CASE units OF
    AxesMoveProcessWidgetUnits.ARCMINUTES:
        unitsText := '$'';
        aziDeg := field_azi_decimal / 60.0;
        eleDeg := field_ele_decimal / 60.0;
        rocDeg := field_roc_decimal / 60.0;
        ronDeg := field_ron_decimal / 60.0;
    AxesMoveProcessWidgetUnits.ARCSECCONDS:
        unitsText := '"';
        aziDeg := field_azi_decimal / 3600.0;
        eleDeg := field_ele_decimal / 3600.0;
        rocDeg := field_roc_decimal / 3600.0;
        ronDeg := field_ron_decimal / 3600.0;
    AxesMoveProcessWidgetUnits.DEGMINSEC:
        unitsText := '';
        aziDeg := DMS_TO_DEG(
            positive := field_azi_sign = AxesDialogSign.DIALOG_PLUS,
            degrees  := field_azi_d,
            minutes  := field_azi_m,
            seconds  := field_azi_s);
        eleDeg := DMS_TO_DEG(
            positive := field_ele_sign = AxesDialogSign.DIALOG_PLUS,
            degrees  := field_ele_d,
            minutes  := field_ele_m,
            seconds  := field_ele_s);
        rocDeg := DMS_TO_DEG(
            positive := field_roc_sign = AxesDialogSign.DIALOG_PLUS,
            degrees  := field_roc_d,
            minutes  := field_roc_m,
            seconds  := field_roc_s);
        ronDeg := DMS_TO_DEG(
            positive := field_ron_sign = AxesDialogSign.DIALOG_PLUS,
            degrees  := field_ron_d,
            minutes  := field_ron_m,
            seconds  := field_ron_s);
    AxesMoveProcessWidgetUnits.DEGREES:
        unitsText := '°';
        aziDeg := field_azi_decimal;
        eleDeg := field_ele_decimal;
        rocDeg := field_roc_decimal;
        ronDeg := field_ron_decimal;
    AxesMoveProcessWidgetUnits.RADIANS:
        unitsText := 'rad';
        aziDeg := RAD_TO_DEG(field_azi_decimal);
        eleDeg := RAD_TO_DEG(field_ele_decimal);
        rocDeg := RAD_TO_DEG(field_roc_decimal);
        ronDeg := RAD_TO_DEG(field_ron_decimal);
END_CASE

END_FUNCTION_BLOCK

// ---- MTCS/Axes/Widgets/AxesManualMoveVelocityWidget.TcPOU
FUNCTION_BLOCK AxesManualMoveVelocityWidget
VAR_INPUT
    field_alphaVelocity : LREAL;
    field_deltaVelocity : LREAL;
    field_units : AxesMoveVelocityUnits;
    label_units : STRING;
    do_start : BOOL;
    do_stop : BOOL;
    
    setAlphaDeltaVelocityStatus : StatusWidget;
END_VAR
VAR_OUTPUT
    alphaTravelledSoFar : AxesAlphaWidget;
    deltaTravelledSoFar : AxesDeltaWidget;
    alphaPerMinute : AxesAlphaWidget;
    deltaPerMinute : AxesDeltaWidget;
END_VAR
VAR_IN_OUT
    ref : Axes;
END_VAR
VAR
END_VAR


setAlphaDeltaVelocityStatus(
    text  := ref.processes.setAlphaDeltaVelocity.actualStatus,
    color := HealthBusyToColor(healthStatus := ref.processes.setAlphaDeltaVelocity.statuses.healthStatus, 
                               busyStatus   := ref.processes.setAlphaDeltaVelocity.statuses.busyStatus));

label_units := AxesMoveVelocityUnitsToString(field_units);
                      
alphaTravelledSoFar(radians := ref.target.alphaTravelled.radians.value);
deltaTravelledSoFar(radians := ref.target.deltaTravelled.radians.value);

alphaPerMinute(radians := ref.target.alphaVelocity.radiansPerSecond.value * 60.0);
deltaPerMinute(radians := ref.target.deltaVelocity.radiansPerSecond.value * 60.0);

IF do_start THEN
    ref.processes.setAlphaDeltaVelocity.request( units := field_units, alphaVelocity := field_alphaVelocity, deltaVelocity := field_deltaVelocity);
    do_start := FALSE;
END_IF

IF do_stop THEN
    ref.processes.setAlphaDeltaVelocity.request( units := AxesMoveVelocityUnits.ARCSECONDS_PER_SECOND, alphaVelocity := 0.0, deltaVelocity := 0.0);
    do_stop := FALSE;
END_IF

END_FUNCTION_BLOCK

// ---- MTCS/Axes/Widgets/AxesManualPositionsWidget.TcPOU
FUNCTION_BLOCK AxesManualPositionsWidget
VAR_INPUT
END_VAR
VAR_OUTPUT
    invisiblePosition0 : BOOL;
    invisiblePosition1 : BOOL;
    invisiblePosition2 : BOOL;
    invisiblePosition3 : BOOL;
    invisiblePosition4 : BOOL;
    invisiblePosition5 : BOOL;
    invisiblePosition6 : BOOL;
    invisiblePosition7 : BOOL;
    invisiblePosition8 : BOOL;
    invisiblePosition9 : BOOL;
    invisiblePosition10 : BOOL;
    invisiblePosition11 : BOOL;
    invisiblePosition12 : BOOL;
    invisiblePosition13 : BOOL;
    invisiblePosition14 : BOOL;
    invisiblePosition15 : BOOL;
    invisiblePosition16 : BOOL;
    invisiblePosition17 : BOOL;
    invisiblePosition18 : BOOL;
    invisiblePosition19 : BOOL;
END_VAR
VAR_IN_OUT
    ref : Axes;
    ref_operatorStatus : OperatorStatus;
END_VAR
VAR
END_VAR

invisiblePosition0 := NOT (ref.config.knownPositions.position0.allowObserver OR ref_operatorStatus.tech) OR ref.config.knownPositions.position0.name = '';
invisiblePosition1 := NOT (ref.config.knownPositions.position1.allowObserver OR ref_operatorStatus.tech) OR ref.config.knownPositions.position1.name = '';
invisiblePosition2 := NOT (ref.config.knownPositions.position2.allowObserver OR ref_operatorStatus.tech) OR ref.config.knownPositions.position2.name = '';
invisiblePosition3 := NOT (ref.config.knownPositions.position3.allowObserver OR ref_operatorStatus.tech) OR ref.config.knownPositions.position3.name = '';
invisiblePosition4 := NOT (ref.config.knownPositions.position4.allowObserver OR ref_operatorStatus.tech) OR ref.config.knownPositions.position4.name = '';
invisiblePosition5 := NOT (ref.config.knownPositions.position5.allowObserver OR ref_operatorStatus.tech) OR ref.config.knownPositions.position5.name = '';
invisiblePosition6 := NOT (ref.config.knownPositions.position6.allowObserver OR ref_operatorStatus.tech) OR ref.config.knownPositions.position6.name = '';
invisiblePosition7 := NOT (ref.config.knownPositions.position7.allowObserver OR ref_operatorStatus.tech) OR ref.config.knownPositions.position7.name = '';
invisiblePosition8 := NOT (ref.config.knownPositions.position8.allowObserver OR ref_operatorStatus.tech) OR ref.config.knownPositions.position8.name = '';
invisiblePosition9 := NOT (ref.config.knownPositions.position9.allowObserver OR ref_operatorStatus.tech) OR ref.config.knownPositions.position9.name = '';
invisiblePosition10 := NOT (ref.config.knownPositions.position10.allowObserver OR ref_operatorStatus.tech) OR ref.config.knownPositions.position10.name = '';
invisiblePosition11 := NOT (ref.config.knownPositions.position11.allowObserver OR ref_operatorStatus.tech) OR ref.config.knownPositions.position11.name = '';
invisiblePosition12 := NOT (ref.config.knownPositions.position12.allowObserver OR ref_operatorStatus.tech) OR ref.config.knownPositions.position12.name = '';
invisiblePosition13 := NOT (ref.config.knownPositions.position13.allowObserver OR ref_operatorStatus.tech) OR ref.config.knownPositions.position13.name = '';
invisiblePosition14 := NOT (ref.config.knownPositions.position14.allowObserver OR ref_operatorStatus.tech) OR ref.config.knownPositions.position14.name = '';
invisiblePosition15 := NOT (ref.config.knownPositions.position15.allowObserver OR ref_operatorStatus.tech) OR ref.config.knownPositions.position15.name = '';
invisiblePosition16 := NOT (ref.config.knownPositions.position16.allowObserver OR ref_operatorStatus.tech) OR ref.config.knownPositions.position16.name = '';
invisiblePosition17 := NOT (ref.config.knownPositions.position17.allowObserver OR ref_operatorStatus.tech) OR ref.config.knownPositions.position17.name = '';
invisiblePosition18 := NOT (ref.config.knownPositions.position18.allowObserver OR ref_operatorStatus.tech) OR ref.config.knownPositions.position18.name = '';
invisiblePosition19 := NOT (ref.config.knownPositions.position19.allowObserver OR ref_operatorStatus.tech) OR ref.config.knownPositions.position19.name = '';

END_FUNCTION_BLOCK

// ---- MTCS/Axes/Widgets/AxesManualMoveAbsoluteWidget.TcPOU
FUNCTION_BLOCK AxesManualMoveAbsoluteWidget
VAR_INPUT
    moveAbsolute : AxesMultiMoveProcessWIdget;
END_VAR
VAR_OUTPUT
END_VAR
VAR_IN_OUT
    ref : Axes;
END_VAR
VAR
END_VAR

moveAbsolute(
    aziDisabled := ref.processes.moveAbsolute.statuses.enabledStatus.disabled OR ref.parts.azi.statuses.poweredStatus.disabled,
    eleDisabled := ref.processes.moveAbsolute.statuses.enabledStatus.disabled OR ref.parts.ele.statuses.poweredStatus.disabled,
    rocDisabled := ref.processes.moveAbsolute.statuses.enabledStatus.disabled OR ref.parts.roc.statuses.poweredStatus.disabled,
    ronDisabled := ref.processes.moveAbsolute.statuses.enabledStatus.disabled OR ref.parts.ron.statuses.poweredStatus.disabled,
    process := ref.processes.moveAbsolute,  
    title := 'Move absolute');

END_FUNCTION_BLOCK

// ---- MTCS/Axes/Widgets/AxesElevationAxisWidget.TcPOU
FUNCTION_BLOCK AxesElevationAxisWidget
VAR_INPUT
    activeTab : AxesElevationAxisTabs;
END_VAR
VAR_OUTPUT
END_VAR
VAR_IN_OUT
    ref : AxesElevationAxis;
    ref_driveChannel : AX52XXDriveChannel;
END_VAR
VAR
	actualStatus : StatusWidget;
    
    processes_powerOnStatus : StatusWidget;
    processes_powerOffStatus : StatusWidget;
    processes_resetStatus : StatusWidget;
    processes_doHomingStatus : StatusWidget;
    processes_unlockBrakeStatus : StatusWidget;
    processes_stopStatus : StatusWidget;
    processes_moveAbsoluteStatus : StatusWidget;
    processes_moveRelativeStatus : StatusWidget;
    processes_moveVelocityStatus : StatusWidget;
    processes_moveOutOfLimitSwitchStatus : StatusWidget;
    
    lidaCommonHealthStatus : HealthStatus;
    lidaCommonBusyStatus   : BusyStatus;
    lidaCommonStatusColor  : StatusColor;
    
    processCommonHealthStatus : HealthStatus;
    processCommonBusyStatus   : BusyStatus;
    processCommonStatusColor  : StatusColor;
    
    
    button_overview         : SubSubSystemButtonWidget('Overview'           , AxesElevationAxisTabs.OVERVIEW);
    button_processes        : SubSubSystemButtonWidget('Processes'          , AxesElevationAxisTabs.PROCESSES);
    button_driveChannel     : SubSubSystemButtonWidget('Drive channel'      , AxesElevationAxisTabs.DRIVE_CHANNEL);   
    button_virtualAxis      : SubSubSystemButtonWidget('Virtual axis'       , AxesElevationAxisTabs.VIRTUAL_AXIS);  
    button_physicalAxis     : SubSubSystemButtonWidget('Physical axis'      , AxesElevationAxisTabs.PHYSICAL_AXIS);  
    button_lidas            : SubSubSystemButtonWidget('LIDAs'              , AxesElevationAxisTabs.LIDAS);
    button_absoluteEncoder  : SubSubSystemButtonWidget('Absolute encoder'   , AxesElevationAxisTabs.ABSOLUTE_ENCODER);
    
    driveChannel    : AX52XXDriveChannelWidget;
    virtualAxis     : AngularAxisWidget;
    physicalAxis    : AngularAxisWidget;
    
    lida1 : IncrementalEncoderWidget;
    lida2 : IncrementalEncoderWidget;
    
    actPos : AxesAngleWidget;
    setPos : AxesAngleWidget;
    targetPos : AxesAngleWidget;
END_VAR


actualStatus(text  := ref.actualStatus,
             color := HealthBusyToColor(healthStatus := ref.statuses.healthStatus, 
                                        busyStatus   := ref.statuses.busyStatus));

processes_powerOffStatus(
    text  := ref.processes.powerOff.actualStatus,
    color := HealthBusyToColor(healthStatus := ref.processes.powerOff.statuses.healthStatus, 
                               busyStatus   := ref.processes.powerOff.statuses.busyStatus));
processes_powerOnStatus(
    text  := ref.processes.powerOn.actualStatus,
    color := HealthBusyToColor(healthStatus := ref.processes.powerOn.statuses.healthStatus, 
                               busyStatus   := ref.processes.powerOn.statuses.busyStatus));
processes_resetStatus(
    text  := ref.processes.reset.actualStatus,
    color := HealthBusyToColor(healthStatus := ref.processes.reset.statuses.healthStatus, 
                               busyStatus   := ref.processes.reset.statuses.busyStatus));
processes_doHomingStatus(
    text  := ref.processes.doHoming.actualStatus,
    color := HealthBusyToColor(healthStatus := ref.processes.doHoming.statuses.healthStatus, 
                               busyStatus   := ref.processes.doHoming.statuses.busyStatus));
processes_unlockBrakeStatus(
    text  := ref.processes.unlockBrake.actualStatus,
    color := HealthBusyToColor(healthStatus := ref.processes.unlockBrake.statuses.healthStatus, 
                               busyStatus   := ref.processes.unlockBrake.statuses.busyStatus));
processes_stopStatus(
    text  := ref.processes.stop.actualStatus,
    color := HealthBusyToColor(healthStatus := ref.processes.stop.statuses.healthStatus, 
                               busyStatus   := ref.processes.stop.statuses.busyStatus));
processes_moveAbsoluteStatus(
    text  := ref.processes.moveAbsolute.actualStatus,
    color := HealthBusyToColor(healthStatus := ref.processes.moveAbsolute.statuses.healthStatus, 
                               busyStatus   := ref.processes.moveAbsolute.statuses.busyStatus));
processes_moveRelativeStatus(
    text  := ref.processes.moveRelative.actualStatus,
    color := HealthBusyToColor(healthStatus := ref.processes.moveRelative.statuses.healthStatus, 
                               busyStatus   := ref.processes.moveRelative.statuses.busyStatus));
processes_moveVelocityStatus(
    text  := ref.processes.moveVelocity.actualStatus,
    color := HealthBusyToColor(healthStatus := ref.processes.moveVelocity.statuses.healthStatus, 
                               busyStatus   := ref.processes.moveVelocity.statuses.busyStatus));
processes_moveOutOfLimitSwitchStatus(
    text  := ref.processes.moveOutOfLimitSwitch.actualStatus,
    color := HealthBusyToColor(healthStatus := ref.processes.moveOutOfLimitSwitch.statuses.healthStatus, 
                               busyStatus   := ref.processes.moveOutOfLimitSwitch.statuses.busyStatus));


driveChannel(ref := ref_driveChannel, name := 'ELE (Drive ELED channel A)');
virtualAxis(baseRef := ref.parts.virtualAxis, ref := ref.parts.virtualAxis);
physicalAxis(baseRef := ref.parts.physicalAxis, ref := ref.parts.physicalAxis);                


lidaCommonHealthStatus(
     isGood :=      ref.parts.lida1.statuses.healthStatus.isGood 
                AND ref.parts.lida2.statuses.healthStatus.isGood,
     hasWarning :=  ref.parts.lida1.statuses.healthStatus.hasWarning 
                 OR ref.parts.lida2.statuses.healthStatus.hasWarning);

lidaCommonBusyStatus(
    isBusy :=      ref.parts.lida1.statuses.busyStatus.isBusy 
                OR ref.parts.lida2.statuses.busyStatus.isBusy);

lidaCommonStatusColor := HealthBusyToColor(healthStatus := lidaCommonHealthStatus, busyStatus := lidaCommonBusyStatus);


processCommonHealthStatus(
     isGood :=      ref.processes.powerOn.statuses.healthStatus.isGood 
                AND ref.processes.powerOff.statuses.healthStatus.isGood
                AND ref.processes.reset.statuses.healthStatus.isGood
                AND ref.processes.doHoming.statuses.healthStatus.isGood
                AND ref.processes.unlockBrake.statuses.healthStatus.isGood
                AND ref.processes.stop.statuses.healthStatus.isGood
                AND ref.processes.moveAbsolute.statuses.healthStatus.isGood
                AND ref.processes.moveRelative.statuses.healthStatus.isGood
                AND ref.processes.moveVelocity.statuses.healthStatus.isGood
                AND ref.processes.moveOutOfLimitSwitch.statuses.healthStatus.isGood,
     hasWarning :=  ref.processes.powerOn.statuses.healthStatus.hasWarning 
                 OR ref.processes.powerOff.statuses.healthStatus.hasWarning
                 OR ref.processes.reset.statuses.healthStatus.hasWarning
                 OR ref.processes.doHoming.statuses.healthStatus.hasWarning
                 OR ref.processes.unlockBrake.statuses.healthStatus.hasWarning
                 OR ref.processes.stop.statuses.healthStatus.hasWarning
                 OR ref.processes.moveAbsolute.statuses.healthStatus.hasWarning
                 OR ref.processes.moveRelative.statuses.healthStatus.hasWarning
                 OR ref.processes.moveVelocity.statuses.healthStatus.hasWarning
                 OR ref.processes.moveOutOfLimitSwitch.statuses.healthStatus.hasWarning);

processCommonBusyStatus(
    isBusy :=      ref.processes.powerOn.statuses.busyStatus.busy 
                 OR ref.processes.powerOff.statuses.busyStatus.busy
                 OR ref.processes.reset.statuses.busyStatus.busy
                 OR ref.processes.doHoming.statuses.busyStatus.busy
                 OR ref.processes.unlockBrake.statuses.busyStatus.busy
                 OR ref.processes.stop.statuses.busyStatus.busy
                 OR ref.processes.moveAbsolute.statuses.busyStatus.busy
                 OR ref.processes.moveRelative.statuses.busyStatus.busy
                 OR ref.processes.moveVelocity.statuses.busyStatus.busy
                 OR ref.processes.moveOutOfLimitSwitch.statuses.busyStatus.busy);

processCommonStatusColor := HealthBusyToColor(healthStatus := processCommonHealthStatus, busyStatus := processCommonBusyStatus);
     

lida1(ref := ref.parts.lida1);
lida2(ref := ref.parts.lida2);

button_overview(        color := actualStatus.color                     , activeTab := activeTab);
button_processes(       color := processCommonStatusColor               , activeTab := activeTab);
button_driveChannel(    color := driveChannel.actualStatus.color        , activeTab := activeTab);
button_virtualAxis(     color := virtualAxis.base.actualStatus.color    , activeTab := activeTab);
button_physicalAxis(    color := physicalAxis.base.actualStatus.color   , activeTab := activeTab);
button_lidas(           color := lidaCommonStatusColor                  , activeTab := activeTab);
button_absoluteEncoder( color := HealthToColor(ref.parts.absoluteEncoder.statuses.healthStatus), activeTab := activeTab);

actPos(degrees := ref.actPos.degrees.value, format := '%d° %.2d$' %04.1f"', showPlus := FALSE, showMinus := TRUE);
setPos(degrees := ref.setPos.degrees.value, format := '%d° %.2d$' %04.1f"', showPlus := FALSE, showMinus := TRUE);
targetPos(degrees := ref.targetPos.degrees.value, format := '%d° %.2d$' %04.1f"', showPlus := FALSE, showMinus := TRUE);

END_FUNCTION_BLOCK

// ---- MTCS/Common/Widgets/SubSubSystemButtonWidget.TcPOU
FUNCTION_BLOCK SubSubSystemButtonWidget EXTENDS SubSystemButtonWidget
VAR_INPUT
END_VAR
VAR_IN_OUT
END_VAR
VAR_OUTPUT
END_VAR
VAR
END_VAR

SUPER^(activeTab := activeTab);

END_FUNCTION_BLOCK

// ---- MTCS/Common/Widgets/SubSystemButtonWidget.TcPOU
FUNCTION_BLOCK SubSystemButtonWidget
VAR_INPUT
    color : StatusColor;
    hideColor : BOOL := FALSE;
END_VAR
VAR_IN_OUT
    activeTab : INT;
END_VAR
VAR_OUTPUT
    name : STRING;
    thisTab : INT;
    colorVisible : BOOL;
    
    activated : BOOL;
    notActivated : BOOL;
    
    isNotGreen : BOOL;
    isNotRed : BOOL;
    isNotBlue : BOOL;
    isNotOrange : BOOL;
    isNotGray : BOOL;
END_VAR
VAR
    do_activate : BOOL;
END_VAR


IF do_activate THEN
    activeTab := thisTab;
    do_activate := FALSE;
END_IF

activated := activeTab = thisTab;
notActivated := NOT activated;

isNotRed    := color.bg <> Colors.RED;
isNotBlue   := color.bg <> Colors.BLUE;
isNotOrange := color.bg <> Colors.ORANGE;
isNotGray   := color.bg <> Colors.GRAY;
isNotGreen  := color.bg <> Colors.GREEN;

METHOD FB_init : BOOL
VAR_INPUT
	bInitRetains : BOOL; // if TRUE, the retain variables are initialized (warm start / cold start)
	bInCopyCode : BOOL;  // if TRUE, the instance afterwards gets moved into the copy code (online change)
    n : STRING;
    tab : INT;
END_VAR
name := n;
thisTab := tab;
END_METHOD

END_FUNCTION_BLOCK

// ---- MTCS/Common/Widgets/AX52XXDriveChannelWidget.TcPOU
FUNCTION_BLOCK AX52XXDriveChannelWidget
VAR_INPUT
    name : STRING;
END_VAR
VAR_OUTPUT
	actualStatus : StatusWidget;
    
    input0 : BOOL;
    input1 : BOOL;
    input2 : BOOL;
    input3 : BOOL;
    input4 : BOOL;
    input5 : BOOL;
    input6 : BOOL;
    input7 : BOOL;
    
    output0 : BOOL;
    output1 : BOOL;
    output2 : BOOL;
    output3 : BOOL;
    output4 : BOOL;
    output5 : BOOL;
    output6 : BOOL;
    output7 : BOOL;
    
	processes_setBrakeStatus : StatusWidget;
	processes_acknowledgeSafetyError : StatusWidget;
END_VAR
VAR
END_VAR
VAR_IN_OUT
	ref : AX52XXDriveChannel;
END_VAR


actualStatus(text  := ref.actualStatus,
             color := HealthBusyToColor(healthStatus := ref.statuses.healthStatus, 
                                        busyStatus   := ref.statuses.busyStatus));
                                        
input0 := ref.digitalInputs.0;          
input1 := ref.digitalInputs.1;          
input2 := ref.digitalInputs.2;          
input3 := ref.digitalInputs.3;          
input4 := ref.digitalInputs.4;          
input5 := ref.digitalInputs.5;          
input6 := ref.digitalInputs.6;          
input7 := ref.digitalInputs.7;
      
output0 := ref.digitalOutputs.0;
output1 := ref.digitalOutputs.1;
output2 := ref.digitalOutputs.2;
output3 := ref.digitalOutputs.3;
output4 := ref.digitalOutputs.4;
output5 := ref.digitalOutputs.5;
output6 := ref.digitalOutputs.6;
output7 := ref.digitalOutputs.7;

processes_setBrakeStatus(text  := ref.processes.setBrake.actualStatus,
                         color := HealthBusyToColor(healthStatus := ref.processes.setBrake.statuses.healthStatus, 
                                                    busyStatus   := ref.processes.setBrake.statuses.busyStatus));
processes_acknowledgeSafetyError(text  := ref.processes.acknowledgeSafetyError.actualStatus,
                         color := HealthBusyToColor(healthStatus := ref.processes.acknowledgeSafetyError.statuses.healthStatus, 
                                                    busyStatus   := ref.processes.acknowledgeSafetyError.statuses.busyStatus));

END_FUNCTION_BLOCK

// ---- MTCS/Common/Widgets/AngularAxisWidget.TcPOU
FUNCTION_BLOCK AngularAxisWidget
VAR_INPUT
END_VAR
VAR_OUTPUT
    positionSymbol : STRING := '°';
    velocitySymbol : STRING := '°/s';
    base : BaseAxisWidget;
END_VAR
VAR_IN_OUT
    baseRef : AngularAxis;
    ref : AngularAxis;
END_VAR
VAR
END_VAR

base(ref := baseRef);

END_FUNCTION_BLOCK

// ---- MTCS/Common/Widgets/BaseAxisWidget.TcPOU
FUNCTION_BLOCK BaseAxisWidget
VAR_INPUT
END_VAR
VAR_OUTPUT
    coupled : BOOL;
    decoupled : BOOL;
	(* widgets *)
	moveAbsoluteProcess : McProcessWidget;
	moveVelocityProcess : McProcessWidget;
	actualStatus : StatusWidget;
END_VAR
VAR_IN_OUT
    ref : BaseAxis;
END_VAR
VAR
END_VAR


coupled := ref.axis_ref.Status.Coupled;
decoupled := NOT coupled;

// update the widgets
moveAbsoluteProcess(process := ref.processes.moveAbsolute);
moveVelocityProcess(process := ref.processes.moveVelocity);
actualStatus(text  := ref.actualStatus,
             color := HealthBusyToColor(healthStatus := ref.statuses.healthStatus, 
                                        busyStatus   := ref.statuses.busyStatus));

END_FUNCTION_BLOCK

// ---- MTCS/Common/Widgets/McProcessWidget.TcPOU
FUNCTION_BLOCK McProcessWidget
VAR_INPUT
END_VAR
VAR_OUTPUT
    actualStatus : StatusWidget;
END_VAR
VAR_IN_OUT
	process : BaseMcProcess;
END_VAR
VAR
END_VAR

actualStatus(text  := process.actualStatus,
             color := HealthBusyToColor(healthStatus := process.statuses.healthStatus,
                                        busyStatus   := process.statuses.busyStatus));

END_FUNCTION_BLOCK

// ---- MTCS/Common/StateMachines/BaseMcProcess.TcPOU
FUNCTION_BLOCK BaseMcProcess EXTENDS SM_BaseMcProcess
VAR_INPUT
END_VAR
VAR_OUTPUT
END_VAR
VAR
	testVar3 : BOOL;
END_VAR

SUPER^();
                                  
IF statuses.healthStatus.good THEN

	IF statuses.busyStatus.idle THEN
		actualStatus := 'Idle';
	ELSIF statuses.busyStatus.busy THEN
		actualStatus := 'Busy';
	ELSE
		actualStatus := '';
	END_IF;

ELSIF statuses.healthStatus.bad THEN
	
	IF statuses.busyStatus.idle THEN
		IF errorId = 0 THEN
			actualStatus := 'Error';
		ELSE
			actualStatus := CONCAT(CONCAT('Error (', UDINT_TO_STRING(errorId)), ')');
		END_IF
	ELSIF statuses.busyStatus.busy THEN
		IF errorId = 0 THEN
			actualStatus := 'Busy and error';
		ELSE
			actualStatus := CONCAT(CONCAT('Busy and error (', UDINT_TO_STRING(errorId)), ')');
		END_IF
	ELSE
		IF errorId = 0 THEN
			actualStatus := 'Error';
		ELSE
			actualStatus := CONCAT(CONCAT('Error (', UDINT_TO_STRING(errorId)), ')');
		END_IF
	END_IF;

ELSE
	actualStatus := '';
END_IF;

END_FUNCTION_BLOCK

// ---- MTCS/Common/StateMachines/BaseAxis.TcPOU
FUNCTION_BLOCK BaseAxis EXTENDS SM_BaseAxis
VAR_INPUT
END_VAR
VAR_OUTPUT
END_VAR
VAR
	_mc_moveAbsolute1         : MC_MoveAbsolute;
	_mc_moveAbsolute2         : MC_MoveAbsolute;
    _moveAbsoluteAlternator   : BOOL;
    _previousMoveAbsolutePosition : LREAL;
    _previousMoveAbsoluteMaxVelocity : LREAL;
    _moveAbsoluteStopping   : BOOL;
    _mc_moveVelocity : MC_MoveVelocity;
    _mc_moveRelative : MC_MoveRelative;
    
	_mc_power : MC_Power;
	_mc_reset : MC_Reset;
	_mc_halt : MC_Halt;
	_mc_halt2 : MC_Halt;
	_mc_gearIn : MC_GearIn;
	_mc_gearOut : MC_GearOut;
    _mc_setPosition : MC_SetPosition;
    _mc_extSetPointGenEnable : MC_ExtSetPointGenEnable;
    _mc_extSetPointGenDisable : MC_ExtSetPointGenDisable;
    _mc_home : MC_Home;
    _mc_jog : MC_Jog;
    
	_powered : BOOL;
    
    _masterAddr : POINTER TO AXIS_REF := 0;
    
    _ctrl_pi_params : ST_CTRL_PI_PARAMS;
    _ctrl_pi : FB_CTRL_PI;
    _mc_moveVelocity1 : MC_MoveVelocity;
    _mc_moveVelocity2 : MC_MoveVelocity;
    
    _mc_writeParameter : MC_WriteParameter;
    _mc_writeBoolParameter : MC_WriteBoolParameter;
    _mc_readParameter : MC_ReadParameter;
    _mc_readBoolParameter : MC_ReadBoolParameter;
    
    
    Kp : LREAL := 1.0;
    Td : LREAL := 0.0;
END_VAR

SUPER^.axis_ref.ReadStatus();

_update();

// command the axis
_powering();
_movingAbsolute();
_movingRelative();
_resetting();
_initializing();
_stopping();
_stoppingParametrized();
_gearIn();
_gearOut();
_setPosition();
_moveVelocity();
_enableExtSetGen();
_disableExtSetGen();
_forceCalibration();
_resetCalibration();

_readParameter();
_readBoolParameter();
_writeParameter();
_writeBoolParameter();

_update();

METHOD _forceCalibration
VAR_INPUT
END_VAR

_mc_home(
    Execute     := processes.forceCalibration.statuses.busyStatus.busy,
    Position    := 0.0,
    HomingMode  := MC_HomingMode.MC_ForceCalibration,
    Axis        := axis_ref);

(* update the health status *)
SUPER^.processes.forceCalibration.statuses.healthStatus(isGood := NOT _mc_home.Error);

(* update the busy status *)
SUPER^.processes.forceCalibration.statuses.busyStatus(isBusy := _mc_home.Busy);

(* update the error ID *)
SUPER^.processes.forceCalibration.errorId := _mc_home.ErrorId;
END_METHOD

METHOD _movingAbsolute
VAR_INPUT
END_VAR
IF processes.moveAbsolute.statuses.busyStatus.busy THEN
	
    // MC_MoveAbsolute is a single command to instruct the axis to go to some position.
    // This position cannot be changed later: the command only does what you initially requested
    // (in other words: it only uses the position at the time of the Execute trigger).
    
    // We don' t want this behaviour, as we would like to be able to change the setpoint
    // position also during positioning. There are many use cases for this behaviour, e.g.:
    //  - you can send corrections to the axis while the position loop is running
    //  - you can change your mind while the positioning is running.
    
    // Therefore, we need 2 MC_MoveAbsolute commands, that abort each other alternatingly.
    // At each PLC cycle, one MC_MoveAbsolute command will be Busy and the other will be
    // CommandAborted. Only when one of them is Done (or Error), the motion has ended.
    
    IF    _previousMoveAbsolutePosition <> processes.moveAbsolute.get.position 
       OR _previousMoveAbsoluteMaxVelocity <> processes.moveAbsolute.get.maxVelocity
    THEN
        _moveAbsoluteAlternator := NOT _moveAbsoluteAlternator;
        _previousMoveAbsolutePosition := processes.moveAbsolute.get.position;
        _previousMoveAbsoluteMaxVelocity := processes.moveAbsolute.get.maxVelocity;
	END_IF
    
    IF _moveAbsoluteAlternator THEN
    
        _mc_moveAbsolute2(Axis := axis_ref, Execute := FALSE);
        
        _mc_moveAbsolute1(
            Axis       := axis_ref,
            Execute    := TRUE,
            Position   := processes.moveAbsolute.get.position,
            Velocity   := processes.moveAbsolute.get.maxVelocity,
            BufferMode := MC_BufferMode.MC_Aborting);
        
        (* update the statuses *)
        processes.moveAbsolute.statuses.healthStatus(isGood := NOT _mc_moveAbsolute1.Error);
        processes.moveAbsolute.errorId := _mc_moveAbsolute1.ErrorId;
        processes.moveAbsolute.statuses.busyStatus(isBusy := _mc_moveAbsolute1.Busy);
    ELSE
        
        _mc_moveAbsolute1(Axis := axis_ref, Execute := FALSE);
        
        _mc_moveAbsolute2(
            Axis       := axis_ref,
            Execute    := TRUE,
            Position   := processes.moveAbsolute.get.position,
            Velocity   := processes.moveAbsolute.get.maxVelocity,
            BufferMode := MC_BufferMode.MC_Aborting);
        
        (* update the statuses *)
        processes.moveAbsolute.statuses.healthStatus(isGood := NOT _mc_moveAbsolute2.Error);
        processes.moveAbsolute.errorId := _mc_moveAbsolute2.ErrorId;
        processes.moveAbsolute.statuses.busyStatus(isBusy := _mc_moveAbsolute2.Busy);
        
	END_IF
	
    (* reset the function blocks if needed *)
    IF processes.moveAbsolute.statuses.busyStatus.idle THEN
        _mc_moveAbsolute1(Axis := axis_ref, Execute := FALSE);
        _mc_moveAbsolute2(Axis := axis_ref, Execute := FALSE);
	END_IF
    
END_IF
END_METHOD

METHOD _writeBoolParameter
VAR_INPUT
END_VAR

_mc_writeBoolParameter(
    Execute         := processes.writeBoolParameter.statuses.busyStatus.busy,
    ParameterNumber := processes.writeBoolParameter.get.parameterNumber,
    Value           := processes.writeBoolParameter.get.value,
    Axis            := axis_ref);

(* update the health status *)
SUPER^.processes.writeBoolParameter.statuses.healthStatus(isGood := NOT _mc_writeBoolParameter.Error);

(* update the busy status *)
SUPER^.processes.writeBoolParameter.statuses.busyStatus(isBusy := _mc_writeBoolParameter.Busy);

(* update the error ID *)
SUPER^.processes.writeBoolParameter.errorId := _mc_writeBoolParameter.ErrorId;
END_METHOD

METHOD _gearIn
VAR_INPUT
END_VAR

IF _masterAddr = 0 THEN
    processes.gearIn.setBad();
    processes.gearIn.setFinished();
ELSE
    _mc_gearIn(
        Execute := processes.gearIn.statuses.busyStatus.busy,
        Master  := _masterAddr^,
        Slave   := axis_ref);
    
    (* update the health status *)
    SUPER^.processes.gearIn.statuses.healthStatus(isGood := NOT _mc_gearIn.Error);
    
    (* update the busy status *)
    SUPER^.processes.gearIn.statuses.busyStatus(isBusy := _mc_gearIn.Busy);
    
    (* update the error ID *)
    SUPER^.processes.gearIn.errorId := _mc_gearIn.ErrorId;
END_IF
END_METHOD

METHOD _moveVelocity
VAR_INPUT
END_VAR

IF processes.moveVelocity.isBusy() THEN
    
    IF NOT processes.moveVelocity.isStarted() THEN
        IF processes.moveVelocity.get.value >= 0 THEN
            _mc_moveVelocity(Execute := FALSE, Axis := axis_ref);
            _mc_moveVelocity(
                Execute      := TRUE,
                Velocity     := ABS(processes.moveVelocity.get.value),
                Acceleration := 0,
                Deceleration := 0,
                Jerk         := 0,
                Direction    := MC_Positive_Direction,
                Axis         := axis_ref);
        ELSE
            _mc_moveVelocity(Execute := FALSE, Axis := axis_ref);
            _mc_moveVelocity(
                Execute      := TRUE,
                Velocity     := ABS(processes.moveVelocity.get.value),
                Acceleration := 0,
                Deceleration := 0,
                Jerk         := 0,
                Direction    := MC_Negative_Direction,
                Axis         := axis_ref);
        END_IF
        processes.moveVelocity.setStarted();
    ELSE
        _mc_moveVelocity(Execute := FALSE, Axis := axis_ref);
	END_IF
    
    (* update the health status *)
    processes.moveVelocity.statuses.healthStatus(isGood := NOT _mc_moveVelocity.Error);
    
    (* update the busy status *)
    processes.moveVelocity.statuses.busyStatus(isBusy := _mc_moveVelocity.Busy AND NOT _mc_moveVelocity.InVelocity);
    
    (* update the error ID *)
    processes.moveVelocity.errorId := _mc_moveVelocity.ErrorId;
    
    
END_IF
END_METHOD

METHOD _readParameter
VAR_INPUT
END_VAR

_mc_readParameter(
    Enable          := processes.readParameter.statuses.busyStatus.busy,
    ParameterNumber := processes.readParameter.get.parameterNumber,
    Axis            := axis_ref,
    Value           => processes.readParameter.value);

(* update the health status *)
SUPER^.processes.readParameter.statuses.healthStatus(isGood := NOT _mc_readParameter.Error);

(* update the busy status *)
SUPER^.processes.readParameter.statuses.busyStatus(isBusy := _mc_readParameter.Busy);

(* update the error ID *)
SUPER^.processes.readParameter.errorId := _mc_readParameter.ErrorId;
END_METHOD

METHOD _stopping
VAR_INPUT
END_VAR

IF processes.stop.statuses.busyStatus.busy THEN
    
    _mc_halt(Execute := TRUE, Axis := axis_ref);
    
    IF _mc_halt.Error OR _mc_halt.Done OR _mc_halt.CommandAborted THEN
        _mc_halt(Execute := FALSE, Axis := axis_ref);
	END_IF
    
    (* update the health status *)
    SUPER^.processes.stop.statuses.healthStatus(isGood := NOT _mc_halt.Error);
    
    (* update the busy status *)
    SUPER^.processes.stop.statuses.busyStatus(isBusy := _mc_halt.Busy);
    
    (* update the error ID *)
    SUPER^.processes.stop.errorId := _mc_halt.ErrorId;
END_IF
END_METHOD

METHOD _resetCalibration
VAR_INPUT
END_VAR

_mc_home(
    Execute     := processes.resetCalibration.statuses.busyStatus.busy,
    Position    := 0.0,
    HomingMode  := MC_HomingMode.MC_ResetCalibration,
    Axis        := axis_ref);

(* update the health status *)
SUPER^.processes.resetCalibration.statuses.healthStatus(isGood := NOT _mc_home.Error);

(* update the busy status *)
SUPER^.processes.resetCalibration.statuses.busyStatus(isBusy := _mc_home.Busy);

(* update the error ID *)
SUPER^.processes.resetCalibration.errorId := _mc_home.ErrorId;
END_METHOD

METHOD _tracking_notworking
VAR_INPUT
END_VAR

VAR
    direction : MC_Direction;
END_VAR
IF processes.moveAbsolute.statuses.busyStatus.busy THEN
	
    IF NOT processes.moveAbsolute.isStarted() THEN
        _mc_moveVelocity1(Axis := axis_ref, Execute := FALSE);
        _mc_moveVelocity2(Axis := axis_ref, Execute := FALSE);
        _ctrl_pi_params.tCtrlCycleTime := GLOBAL.config.PLC_CTRL_TIME;
        _ctrl_pi_params.tTaskCycleTime := GLOBAL.config.PLC_TASK_TIME;
        processes.moveAbsolute.setStarted();
    END_IF

    _ctrl_pi_params.fKp := Kp;
    _ctrl_pi_params.tTn := LREAL_TO_TIME(Td); //ms
    _ctrl_pi_params.fOutMaxLimit :=  processes.moveAbsolute.get.maxVelocity;
    _ctrl_pi_params.fOutMinLimit := -processes.moveAbsolute.get.maxVelocity;
    
    _ctrl_pi(
        fSetpointValue := processes.moveAbsolute.get.position,
        fActualValue   := axis_ref.NcToPlc.ActPos,
        fManSyncValue  := 0.0,
        bSync          := FALSE,
        eMode          := eCTRL_MODE_ACTIVE,
        bHold          := FALSE,
        stParams       := _ctrl_pi_params);
    
    IF _ctrl_pi.fOut > 0 THEN
        direction := MC_Positive_Direction;
    ELSE
        direction := MC_Negative_Direction;
	END_IF
    
    _moveAbsoluteAlternator := NOT _moveAbsoluteAlternator;
    
    _moveAbsoluteStopping := ABS(processes.moveAbsolute.get.position - axis_ref.NcToPlc.ActPos) < 0.001
                             OR _mc_moveVelocity1.Error 
                             OR _mc_moveVelocity2.Error
                             OR (_mc_moveVelocity1.CommandAborted AND _mc_moveVelocity2.CommandAborted);
    
    IF _moveAbsoluteStopping THEN
        _mc_halt(Execute := TRUE, Axis := axis_ref);
        IF _mc_halt.Done THEN
            _mc_halt(Execute := FALSE, Axis := axis_ref);
            processes.moveAbsolute.setGood();
            processes.moveAbsolute.setFinished();
        ELSIF _mc_halt.Error OR _mc_halt.CommandAborted THEN
            _mc_halt(Execute := FALSE, Axis := axis_ref);
            processes.moveAbsolute.setBad();
            processes.moveAbsolute.setFinished();
		END_IF
    ELSIF _moveAbsoluteAlternator THEN
        _mc_moveVelocity2(Axis := axis_ref, Execute := FALSE);
        _mc_moveVelocity1(
            Execute      := TRUE,
            Velocity     := ABS(_ctrl_pi.fOut),
            Acceleration := 0,
            Deceleration := 0,
            Jerk         := 0,
            Direction    := direction,
            BufferMode := MC_BufferMode.MC_Aborting,
            Axis         := axis_ref);
            
            (* update the statuses *)
            //processes.moveAbsolute.statuses.busyStatus(isBusy := _mc_moveVelocity1.Busy);
            processes.moveAbsolute.statuses.healthStatus(isGood := NOT _mc_moveVelocity1.Error);
            processes.moveAbsolute.errorId := _mc_moveVelocity1.ErrorId;
    ELSE
        _mc_moveVelocity1(Axis := axis_ref, Execute := FALSE);
        _mc_moveVelocity2(
            Execute      := TRUE,
            Velocity     := ABS(_ctrl_pi.fOut),
            Acceleration := 0,
            Deceleration := 0,
            Jerk         := 0,
            Direction    := direction,
            BufferMode := MC_BufferMode.MC_Aborting,
            Axis         := axis_ref);
            
            (* update the statuses *)
            //processes.moveAbsolute.statuses.busyStatus(isBusy := _mc_moveVelocity2.Busy);
            processes.moveAbsolute.statuses.healthStatus(isGood := NOT _mc_moveVelocity2.Error);
            processes.moveAbsolute.errorId := _mc_moveVelocity2.ErrorId;
	END_IF
    
ELSE
    
    _ctrl_pi(eMode := eCTRL_MODE_RESET, stParams := _ctrl_pi_params);
    
END_IF
END_METHOD

METHOD _setPosition
VAR_INPUT
END_VAR

_mc_setPosition(
    Execute  := processes.setPosition.statuses.busyStatus.busy,
    Position := processes.setPosition.get.value,
    Mode     := FALSE,
    Axis     := axis_ref);

(* update the health status *)
SUPER^.processes.setPosition.statuses.healthStatus(isGood := NOT _mc_setPosition.Error);

(* update the busy status *)
SUPER^.processes.setPosition.statuses.busyStatus(isBusy := _mc_setPosition.Busy);

(* update the error ID *)
SUPER^.processes.setPosition.errorId := _mc_setPosition.ErrorId;
END_METHOD

METHOD _readBoolParameter
VAR_INPUT
END_VAR

_mc_readBoolParameter(
    Enable          := processes.readBoolParameter.statuses.busyStatus.busy,
    ParameterNumber := processes.readBoolParameter.get.parameterNumber,
    Axis            := axis_ref,
    Value           => processes.readBoolParameter.value);

(* update the health status *)
SUPER^.processes.readBoolParameter.statuses.healthStatus(isGood := NOT _mc_readBoolParameter.Error);

(* update the busy status *)
SUPER^.processes.readBoolParameter.statuses.busyStatus(isBusy := _mc_readBoolParameter.Busy);

(* update the error ID *)
SUPER^.processes.readBoolParameter.errorId := _mc_readBoolParameter.ErrorId;
END_METHOD

METHOD _update
VAR_INPUT
END_VAR
SUPER^();

IF statuses.healthStatus.good THEN
    IF statuses.busyStatus.idle THEN
        IF statuses.poweredStatus.enabled THEN
            actualStatus := 'Enabled';
        ELSIF statuses.poweredStatus.disabled THEN
            actualStatus := 'Disabled';
        ELSE
            actualStatus := 'Idle';
		END_IF
    ELSIF statuses.busyStatus.busy THEN
        IF statuses.motionStatus.forward THEN
            actualStatus := 'Moving forward';
        ELSIF statuses.motionStatus.backward THEN
            actualStatus := 'Moving backward';
        ELSIF statuses.motionStatus.standstill THEN
            actualStatus := 'Standing still';
        ELSE
            actualStatus := 'Busy';
		END_IF
    ELSE
        actualStatus := 'Good';
    END_IF
ELSIF statuses.healthStatus.bad THEN
    IF axis_ref.Status.ErrorId = 16992 THEN
        actualStatus := 'Controller not enabled!';
    ELSIF axis_ref.Status.ErrorId = 18000 THEN
        actualStatus := 'Drive not ready!';
    ELSE
        actualStatus := CONCAT(CONCAT('Error (id: ', UDINT_TO_STRING(axis_ref.Status.ErrorId)), ')');
	END_IF
ELSE
    actualStatus := '';
END_IF
END_METHOD

METHOD _enableExtSetGen
VAR_INPUT
END_VAR
_mc_extSetPointGenEnable(
	Axis    := axis_ref,
	Execute := processes.enableExtSetGen.statuses.busyStatus.busy);

(* update the health status *)
SUPER^.processes.enableExtSetGen.statuses.healthStatus(isGood := NOT _mc_extSetPointGenEnable.Error);

(* update the busy status *)
SUPER^.processes.enableExtSetGen.statuses.busyStatus(isBusy := _mc_extSetPointGenEnable.Busy);

(* update the error ID *)
SUPER^.processes.enableExtSetGen.errorId := _mc_extSetPointGenEnable.ErrorId;
END_METHOD

METHOD _initializing
VAR_INPUT
END_VAR
IF processes.initialize.statuses.busyStatus.busy THEN
    
	IF processes.initialize.statuses.startedStatus.notStarted THEN
		processes.reset.start();
		processes.initialize.setStarted();
	END_IF
    
    processes.initialize.statuses.busyStatus(isBusy := processes.reset.statuses.busyStatus.busy);
    processes.initialize.statuses.healthStatus(isGood := processes.reset.statuses.healthStatus.good);
    
    
ELSE
    // done
	processes.initialize.setFinished();
END_IF
END_METHOD

METHOD _disableExtSetGen
VAR_INPUT
END_VAR
_mc_extSetPointGenDisable(
	Axis    := axis_ref,
	Execute := processes.disableExtSetGen.statuses.busyStatus.busy);

(* update the health status *)
SUPER^.processes.disableExtSetGen.statuses.healthStatus(isGood := NOT _mc_extSetPointGenDisable.Error);

(* update the busy status *)
SUPER^.processes.disableExtSetGen.statuses.busyStatus(isBusy := _mc_extSetPointGenDisable.Busy);

(* update the error ID *)
SUPER^.processes.disableExtSetGen.errorId := _mc_extSetPointGenDisable.ErrorId;
END_METHOD

METHOD _writeParameter
VAR_INPUT
END_VAR

_mc_writeParameter(
    Execute         := processes.writeParameter.statuses.busyStatus.busy,
    ParameterNumber := processes.writeParameter.get.parameterNumber,
    Value           := processes.writeParameter.get.value,
    Axis            := axis_ref);

(* update the health status *)
SUPER^.processes.writeParameter.statuses.healthStatus(isGood := NOT _mc_writeParameter.Error);

(* update the busy status *)
SUPER^.processes.writeParameter.statuses.busyStatus(isBusy := _mc_writeParameter.Busy);

(* update the error ID *)
SUPER^.processes.writeParameter.errorId := _mc_writeParameter.ErrorId;
END_METHOD

METHOD _resetting
VAR_INPUT
END_VAR
_mc_reset(
	Axis    := axis_ref,
	Execute := processes.reset.statuses.busyStatus.busy);

(* update the health status *)
SUPER^.processes.reset.statuses.healthStatus(isGood := NOT _mc_reset.Error);

(* update the busy status *)
SUPER^.processes.reset.statuses.busyStatus(isBusy := _mc_reset.Busy);

(* update the error ID *)
SUPER^.processes.reset.errorId := _mc_reset.ErrorId;
END_METHOD

METHOD configureMaster
VAR_INPUT
    masterAddr : POINTER TO AXIS_REF;
END_VAR
_masterAddr := masterAddr;
END_METHOD

METHOD _powering
VAR_INPUT
END_VAR
VAR
	enablePower : BOOL;
END_VAR
(* The user can power on/off the axis via the command 'power' of SM_NcSimpleAxis.
   The MC_Power function block however isn't a "command" that can be executed via an Execute trigger,
   but instead it's a function block that requires a "continuous" flag which is either set TRUE or FALSE.
   Therefore, we only execute this MC_Power function block when our command is busy. *)
IF processes.power.statuses.busyStatus.busy THEN
	(* call the MC FB *)
	_mc_power(
		Axis 			:= axis_ref,
		Enable 			:= processes.power.get.enable,
		Enable_Positive := processes.power.get.enable,
		Enable_Negative := processes.power.get.enable);

	(* update the health status *)
	processes.power.statuses.healthStatus(isGood := NOT _mc_power.Error);
	
	(* update the busy status *)
    IF _mc_power.Error THEN
        processes.power.setBad();
        processes.power.setFinished();
    ELSIF _mc_power.Enable THEN
        processes.power.setGood();
        IF _mc_power.Status THEN
            processes.power.setFinished();
        ELSE
            processes.power.setBusy();
		END_IF
    ELSE
        processes.power.setGood();
        IF _mc_power.Busy THEN
            processes.power.setBusy();
        ELSE
            processes.power.setFinished();
		END_IF
	END_IF
	
	(* update the error ID *)
	SUPER^.processes.power.errorId := _mc_power.ErrorId;
END_IF
END_METHOD

METHOD _stoppingParametrized
VAR_INPUT
END_VAR

IF processes.stopParametrized.statuses.busyStatus.busy THEN
    
    _mc_halt2(Execute := TRUE, Deceleration := processes.stopParametrized.get.deceleration, Jerk := processes.stopParametrized.get.jerk, Axis := axis_ref);
    
    IF _mc_halt2.Error OR _mc_halt2.Done OR _mc_halt2.CommandAborted THEN
        _mc_halt2(Execute := FALSE, Axis := axis_ref);
	END_IF
    
    (* update the health status *)
    SUPER^.processes.stopParametrized.statuses.healthStatus(isGood := NOT _mc_halt2.Error);
    
    (* update the busy status *)
    SUPER^.processes.stopParametrized.statuses.busyStatus(isBusy := _mc_halt2.Busy);
    
    (* update the error ID *)
    SUPER^.processes.stopParametrized.errorId := _mc_halt2.ErrorId;
END_IF
END_METHOD

METHOD setPositionCorrection
VAR_INPUT
    positionCorrection : LREAL;
END_VAR
axis_ref.PlcToNc.PositionCorrection := positionCorrection;
END_METHOD

METHOD _movingRelative
VAR_INPUT
END_VAR

IF processes.moveRelative.isBusy() THEN
    
    IF NOT processes.moveRelative.isStarted() THEN
        _mc_moveRelative(Execute := FALSE, Axis := axis_ref);
        _mc_moveRelative(
            Execute      := TRUE,
            Distance     := processes.moveRelative.get.distance,
            Velocity     := processes.moveRelative.get.maxVelocity,
            Acceleration := 0,
            Deceleration := 0,
            Jerk         := 0,
            Axis         := axis_ref);
        processes.moveRelative.setStarted();
    ELSE
        _mc_moveRelative(Execute := FALSE, Axis := axis_ref);
	END_IF
    
    (* update the health status *)
    processes.moveRelative.statuses.healthStatus(isGood := NOT _mc_moveRelative.Error);
    
    (* update the error ID *)
    processes.moveRelative.errorId := _mc_moveRelative.ErrorId;
    
    (* update the busy status *)
    processes.moveRelative.statuses.busyStatus(isBusy := _mc_moveRelative.Busy AND NOT _mc_moveRelative.Done);
    
    
END_IF
END_METHOD

METHOD _gearOut
VAR_INPUT
END_VAR
_mc_gearOut(
    Execute := processes.gearOut.statuses.busyStatus.busy,
    Slave   := axis_ref);

(* update the health status *)
SUPER^.processes.gearOut.statuses.healthStatus(isGood := NOT _mc_gearOut.Error);

(* update the busy status *)
SUPER^.processes.gearOut.statuses.busyStatus(isBusy := _mc_gearOut.Busy);

(* update the error ID *)
SUPER^.processes.gearOut.errorId := _mc_gearOut.ErrorId;
END_METHOD

METHOD jog
VAR_INPUT
    forward : BOOL;
    backwards : BOOL;
    velocity : LREAL;
    acceleration : LREAL;
    deceleration : LREAL;
    
    
END_VAR
isJogEnabled :=  isEnabled 
    AND (statuses.busyStatus.idle OR forward OR backwards)
    AND (statuses.healthStatus.good)
    AND statuses.poweredStatus.enabled;
    
IF isJogEnabled THEN
    
    _mc_jog(
        JogForward := forward,
        JogBackwards := backwards,
        Mode := E_JogMode.MC_JOGMODE_CONTINOUS,
        Position := 0.0,
        Velocity := velocity,
        Acceleration := acceleration,
        Deceleration := deceleration,
        Axis := axis_ref);
ELSE
    

    _mc_jog(
        JogForward := FALSE,
        JogBackwards := FALSE,
        Mode := E_JogMode.MC_JOGMODE_CONTINOUS,
        Position := 0.0,
        Velocity := velocity,
        Acceleration := acceleration,
        Deceleration := deceleration,
        Axis := axis_ref);

END_IF
END_METHOD

END_FUNCTION_BLOCK

// ---- MTCS/Common/Widgets/IncrementalEncoderWidget.TcPOU
FUNCTION_BLOCK IncrementalEncoderWidget
VAR_INPUT
END_VAR
VAR_OUTPUT
END_VAR
VAR_IN_OUT
    ref : IncrementalEncoder;
END_VAR
VAR
	actualStatus : StatusWidget;
END_VAR

actualStatus(text := ref.actualStatus, 
             color := HealthBusyToColor(healthStatus := ref.statuses.healthStatus, 
                                        busyStatus := ref.statuses.busyStatus));

END_FUNCTION_BLOCK

// ---- MTCS/Common/HelperCode/HealthToColor.TcPOU
FUNCTION HealthToColor : StatusColor
VAR_IN_OUT
    healthStatus : HealthStatus;
END_VAR
VAR_OUTPUT
END_VAR
VAR
END_VAR

IF healthStatus.good THEN
    HealthToColor.fg := Colors.BLACK;
    HealthToColor.bg := Colors.GREEN;
ELSIF healthStatus.bad THEN
	HealthToColor.fg := Colors.WHITE;
	HealthToColor.bg := Colors.RED;
ELSIF healthStatus.warning THEN
	HealthToColor.fg := Colors.WHITE;
	HealthToColor.bg := Colors.ORANGE;
ELSE
	HealthToColor.fg := Colors.BLACK;
	HealthToColor.bg := Colors.GRAY;
END_IF

END_FUNCTION

// ---- MTCS/Axes/Widgets/AxesAxesWidget.TcPOU
FUNCTION_BLOCK AxesAxesWidget
VAR_INPUT
    activeTab : AxesAxesTabs;
END_VAR
VAR_OUTPUT
    commonStatusColor : StatusColor;
END_VAR
VAR_IN_OUT
	ref_azi : AxesAzimuthAxis;
	ref_ele : AxesElevationAxis;
	ref_roc : AxesRotationAxis;
	ref_ron : AxesRotationAxis;
    ref_io  : AxesIO;
    //ref_fw  : TODO
END_VAR
VAR    
    button_azi : SubSubSystemButtonWidget('AZI', AxesAxesTabs.AZI);      
    button_ele : SubSubSystemButtonWidget('ELE', AxesAxesTabs.ELE);      
    button_roc : SubSubSystemButtonWidget('ROC', AxesAxesTabs.ROC);      
    button_ron : SubSubSystemButtonWidget('RON', AxesAxesTabs.RON);      
    button_fw  : SubSubSystemButtonWidget('FW' , AxesAxesTabs.FW);      

    azi : AxesAzimuthAxisWidget;
    ele : AxesElevationAxisWidget;
    roc : AxesRotationAxisWidget;
    ron : AxesRotationAxisWidget;
    //fw : AxesPositioningAxisWidget;
    
    commonHealthStatus : HealthStatus;
    commonBusyStatus : BusyStatus;
    
END_VAR

azi(ref := ref_azi, ref_aziDriveChannel := ref_io.parts.aziDrive.parts.channelA, ref_ablDriveChannel := ref_io.parts.ablDrive.parts.channelA);
ele(ref := ref_ele, ref_driveChannel := ref_io.parts.eleDrive.parts.channelA);
roc(ref := ref_roc, ref_driveChannel := ref_io.parts.aziDrive.parts.channelB, axisTitle := 'Rotator Cas.'   , driveChannelTitle := 'ROC (Drive AZID channel B)');
ron(ref := ref_ron, ref_driveChannel := ref_io.parts.ablDrive.parts.channelB, axisTitle := 'Rotator Nas.', driveChannelTitle := 'RON (Drive ABLD channel B)');

button_azi(activeTab := activeTab, color := azi.actualStatus.color);
button_ele(activeTab := activeTab, color := ele.actualStatus.color);
button_roc(activeTab := activeTab, color := roc.actualStatus.color);
button_ron(activeTab := activeTab, color := ron.actualStatus.color);
//button_fw( activeTab := activeTab, color := fw.actualStatus.color);

commonHealthStatus(
     isGood :=      ref_azi.statuses.healthStatus.isGood 
                AND ref_ele.statuses.healthStatus.isGood
                AND ref_roc.statuses.healthStatus.isGood
                AND ref_ron.statuses.healthStatus.isGood,
     hasWarning :=  ref_azi.statuses.healthStatus.hasWarning 
                 OR ref_ele.statuses.healthStatus.hasWarning 
                 OR ref_roc.statuses.healthStatus.hasWarning 
                 OR ref_ron.statuses.healthStatus.hasWarning);
                         
commonBusyStatus(
     isBusy :=    ref_azi.statuses.busyStatus.busy 
               OR ref_ele.statuses.busyStatus.busy 
               OR ref_roc.statuses.busyStatus.busy 
               OR ref_ron.statuses.busyStatus.busy);

commonStatusColor := HealthBusyToColor(
                healthStatus := commonHealthStatus,
                busyStatus := commonBusyStatus);

END_FUNCTION_BLOCK

// ---- MTCS/Axes/Widgets/AxesAzimuthAxisWidget.TcPOU
FUNCTION_BLOCK AxesAzimuthAxisWidget
VAR_INPUT
    activeTab : AxesAzimuthAxisTabs;
END_VAR
VAR_OUTPUT
END_VAR
VAR_IN_OUT
    ref : AxesAzimuthAxis;
    ref_aziDriveChannel : AX52XXDriveChannel;
    ref_ablDriveChannel : AX52XXDriveChannel;
END_VAR
VAR
	actualStatus : StatusWidget;
    
    processes_powerOnStatus : StatusWidget;
    processes_powerOffStatus : StatusWidget;
    processes_resetStatus : StatusWidget;
    processes_doHomingStatus : StatusWidget;
    processes_unlockBrakeStatus : StatusWidget;
    processes_stopStatus : StatusWidget;
    processes_moveAbsoluteStatus : StatusWidget;
    processes_moveRelativeStatus : StatusWidget;
    processes_moveVelocityStatus : StatusWidget;
    processes_moveOutOfLimitSwitchStatus : StatusWidget;
    
    lidaCommonHealthStatus : HealthStatus;
    lidaCommonBusyStatus   : BusyStatus;
    lidaCommonStatusColor  : StatusColor;
    
    processCommonHealthStatus : HealthStatus;
    processCommonBusyStatus   : BusyStatus;
    processCommonStatusColor  : StatusColor;
    
    button_overview         : SubSubSystemButtonWidget('Overview'           , AxesAzimuthAxisTabs.OVERVIEW);
    button_processes        : SubSubSystemButtonWidget('Processes'          , AxesAzimuthAxisTabs.PROCESSES);
    button_aziDriveChannel  : SubSubSystemButtonWidget('AZI drive channel'  , AxesAzimuthAxisTabs.AZI_DRIVE_CHANNEL);   
    button_ablDriveChannel  : SubSubSystemButtonWidget('ABL drive channel'  , AxesAzimuthAxisTabs.ABL_DRIVE_CHANNEL);   
    button_virtualAxis      : SubSubSystemButtonWidget('Virtual axis'       , AxesAzimuthAxisTabs.VIRTUAL_AXIS);  
    button_physicalAxis     : SubSubSystemButtonWidget('Physical axis'      , AxesAzimuthAxisTabs.PHYSICAL_AXIS);  
    button_ablAxis          : SubSubSystemButtonWidget('ABL axis'           , AxesAzimuthAxisTabs.ABL_AXIS);
    button_lidas            : SubSubSystemButtonWidget('LIDAs'              , AxesAzimuthAxisTabs.LIDAS);
    button_absoluteEncoder  : SubSubSystemButtonWidget('Absolute encoder'   , AxesAzimuthAxisTabs.ABSOLUTE_ENCODER);
    
    aziDriveChannel : AX52XXDriveChannelWidget;
    ablDriveChannel : AX52XXDriveChannelWidget;
    virtualAxis     : AngularAxisWidget;
    physicalAxis    : AngularAxisWidget;
    ablAxis         : AngularAxisWidget;
    
    lida1 : IncrementalEncoderWidget;
    lida2 : IncrementalEncoderWidget;
    lida3 : IncrementalEncoderWidget;
    lida4 : IncrementalEncoderWidget;
    
    actPos : AxesAngleWidget;
    setPos : AxesAngleWidget;
    targetPos : AxesAngleWidget;
END_VAR


actualStatus(text  := ref.actualStatus,
             color := HealthBusyToColor(healthStatus := ref.statuses.healthStatus, 
                                        busyStatus   := ref.statuses.busyStatus));

processes_powerOffStatus(
    text  := ref.processes.powerOff.actualStatus,
    color := HealthBusyToColor(healthStatus := ref.processes.powerOff.statuses.healthStatus, 
                               busyStatus   := ref.processes.powerOff.statuses.busyStatus));
processes_powerOnStatus(
    text  := ref.processes.powerOn.actualStatus,
    color := HealthBusyToColor(healthStatus := ref.processes.powerOn.statuses.healthStatus, 
                               busyStatus   := ref.processes.powerOn.statuses.busyStatus));
processes_resetStatus(
    text  := ref.processes.reset.actualStatus,
    color := HealthBusyToColor(healthStatus := ref.processes.reset.statuses.healthStatus, 
                               busyStatus   := ref.processes.reset.statuses.busyStatus));
processes_doHomingStatus(
    text  := ref.processes.doHoming.actualStatus,
    color := HealthBusyToColor(healthStatus := ref.processes.doHoming.statuses.healthStatus, 
                               busyStatus   := ref.processes.doHoming.statuses.busyStatus));
processes_unlockBrakeStatus(
    text  := ref.processes.unlockBrake.actualStatus,
    color := HealthBusyToColor(healthStatus := ref.processes.unlockBrake.statuses.healthStatus, 
                               busyStatus   := ref.processes.unlockBrake.statuses.busyStatus));
processes_stopStatus(
    text  := ref.processes.stop.actualStatus,
    color := HealthBusyToColor(healthStatus := ref.processes.stop.statuses.healthStatus, 
                               busyStatus   := ref.processes.stop.statuses.busyStatus));
processes_moveAbsoluteStatus(
    text  := ref.processes.moveAbsolute.actualStatus,
    color := HealthBusyToColor(healthStatus := ref.processes.moveAbsolute.statuses.healthStatus, 
                               busyStatus   := ref.processes.moveAbsolute.statuses.busyStatus));
processes_moveRelativeStatus(
    text  := ref.processes.moveRelative.actualStatus,
    color := HealthBusyToColor(healthStatus := ref.processes.moveRelative.statuses.healthStatus, 
                               busyStatus   := ref.processes.moveRelative.statuses.busyStatus));
processes_moveVelocityStatus(
    text  := ref.processes.moveVelocity.actualStatus,
    color := HealthBusyToColor(healthStatus := ref.processes.moveVelocity.statuses.healthStatus, 
                               busyStatus   := ref.processes.moveVelocity.statuses.busyStatus));
processes_moveOutOfLimitSwitchStatus(
    text  := ref.processes.moveOutOfLimitSwitch.actualStatus,
    color := HealthBusyToColor(healthStatus := ref.processes.moveOutOfLimitSwitch.statuses.healthStatus, 
                               busyStatus   := ref.processes.moveOutOfLimitSwitch.statuses.busyStatus));


aziDriveChannel(ref := ref_aziDriveChannel, name := 'AZI (Drive AZID channel A)');
ablDriveChannel(ref := ref_ablDriveChannel, name := 'ABL (Drive ABLD channel A)');
virtualAxis(baseRef := ref.parts.virtualAxis, ref := ref.parts.virtualAxis);
physicalAxis(baseRef := ref.parts.physicalAxis, ref := ref.parts.physicalAxis);
ablAxis(baseRef := ref.parts.ablAxis, ref := ref.parts.ablAxis);


lidaCommonHealthStatus(
     isGood :=      ref.parts.lida1.statuses.healthStatus.isGood 
                AND ref.parts.lida2.statuses.healthStatus.isGood
                AND ref.parts.lida3.statuses.healthStatus.isGood
                AND ref.parts.lida4.statuses.healthStatus.isGood,
     hasWarning :=  ref.parts.lida1.statuses.healthStatus.hasWarning 
                 OR ref.parts.lida2.statuses.healthStatus.hasWarning 
                 OR ref.parts.lida3.statuses.healthStatus.hasWarning 
                 OR ref.parts.lida4.statuses.healthStatus.hasWarning);

lidaCommonBusyStatus(
    isBusy :=      ref.parts.lida1.statuses.busyStatus.isBusy 
                OR ref.parts.lida2.statuses.busyStatus.isBusy
                OR ref.parts.lida3.statuses.busyStatus.isBusy
                OR ref.parts.lida4.statuses.busyStatus.isBusy);

lidaCommonStatusColor := HealthBusyToColor(healthStatus := lidaCommonHealthStatus, busyStatus := lidaCommonBusyStatus);
     


processCommonHealthStatus(
     isGood :=      ref.processes.powerOn.statuses.healthStatus.isGood 
                AND ref.processes.powerOff.statuses.healthStatus.isGood
                AND ref.processes.reset.statuses.healthStatus.isGood
                AND ref.processes.doHoming.statuses.healthStatus.isGood
                AND ref.processes.unlockBrake.statuses.healthStatus.isGood
                AND ref.processes.stop.statuses.healthStatus.isGood
                AND ref.processes.moveAbsolute.statuses.healthStatus.isGood
                AND ref.processes.moveRelative.statuses.healthStatus.isGood
                AND ref.processes.moveVelocity.statuses.healthStatus.isGood
                AND ref.processes.moveOutOfLimitSwitch.statuses.healthStatus.isGood,
     hasWarning :=  ref.processes.powerOn.statuses.healthStatus.hasWarning 
                 OR ref.processes.powerOff.statuses.healthStatus.hasWarning
                 OR ref.processes.reset.statuses.healthStatus.hasWarning
                 OR ref.processes.doHoming.statuses.healthStatus.hasWarning
                 OR ref.processes.unlockBrake.statuses.healthStatus.hasWarning
                 OR ref.processes.stop.statuses.healthStatus.hasWarning
                 OR ref.processes.moveAbsolute.statuses.healthStatus.hasWarning
                 OR ref.processes.moveRelative.statuses.healthStatus.hasWarning
                 OR ref.processes.moveVelocity.statuses.healthStatus.hasWarning
                 OR ref.processes.moveOutOfLimitSwitch.statuses.healthStatus.hasWarning);

processCommonBusyStatus(
    isBusy :=      ref.processes.powerOn.statuses.busyStatus.busy 
                 OR ref.processes.powerOff.statuses.busyStatus.busy
                 OR ref.processes.reset.statuses.busyStatus.busy
                 OR ref.processes.doHoming.statuses.busyStatus.busy
                 OR ref.processes.unlockBrake.statuses.busyStatus.busy
                 OR ref.processes.stop.statuses.busyStatus.busy
                 OR ref.processes.moveAbsolute.statuses.busyStatus.busy
                 OR ref.processes.moveRelative.statuses.busyStatus.busy
                 OR ref.processes.moveVelocity.statuses.busyStatus.busy
                 OR ref.processes.moveOutOfLimitSwitch.statuses.busyStatus.busy);

processCommonStatusColor := HealthBusyToColor(healthStatus := processCommonHealthStatus, busyStatus := processCommonBusyStatus);
     

lida1(ref := ref.parts.lida1);
lida2(ref := ref.parts.lida2);
lida3(ref := ref.parts.lida3);
lida4(ref := ref.parts.lida4);

button_overview(        color := actualStatus.color                     , activeTab := activeTab);
button_processes(       color := processCommonStatusColor               , activeTab := activeTab);
button_aziDriveChannel( color := aziDriveChannel.actualStatus.color     , activeTab := activeTab);
button_ablDriveChannel( color := ablDriveChannel.actualStatus.color     , activeTab := activeTab);
button_virtualAxis(     color := virtualAxis.base.actualStatus.color    , activeTab := activeTab);
button_physicalAxis(    color := physicalAxis.base.actualStatus.color   , activeTab := activeTab);
button_ablAxis(         color := ablAxis.base.actualStatus.color        , activeTab := activeTab);
button_lidas(           color := lidaCommonStatusColor                  , activeTab := activeTab);
button_absoluteEncoder( color := HealthToColor(ref.parts.absoluteEncoder.statuses.healthStatus), activeTab := activeTab);

actPos(degrees := ref.actPos.degrees.value, format := '%d° %.2d$' %04.1f"', showPlus := FALSE, showMinus := TRUE);
setPos(degrees := ref.setPos.degrees.value, format := '%d° %.2d$' %04.1f"', showPlus := FALSE, showMinus := TRUE);
targetPos(degrees := ref.targetPos.degrees.value, format := '%d° %.2d$' %04.1f"', showPlus := FALSE, showMinus := TRUE);

END_FUNCTION_BLOCK

// ---- MTCS/Axes/Widgets/AxesRotationAxisWidget.TcPOU
FUNCTION_BLOCK AxesRotationAxisWidget
VAR_INPUT
    activeTab : AxesRotationAxisTabs;
    axisTitle : STRING;
    driveChannelTitle : STRING;
END_VAR
VAR_OUTPUT
END_VAR
VAR_IN_OUT
    ref : AxesRotationAxis;
    ref_driveChannel : AX52XXDriveChannel;
END_VAR
VAR
	actualStatus : StatusWidget;
    
    processes_powerOnStatus : StatusWidget;
    processes_powerOffStatus : StatusWidget;
    processes_resetStatus : StatusWidget;
    processes_stopStatus : StatusWidget;
    processes_moveAbsoluteStatus : StatusWidget;
    processes_moveRelativeStatus : StatusWidget;
    processes_moveVelocityStatus : StatusWidget;
    processes_moveOutOfLimitSwitchStatus : StatusWidget;
    
    processCommonHealthStatus : HealthStatus;
    processCommonBusyStatus   : BusyStatus;
    processCommonStatusColor  : StatusColor;
    
    
    button_overview         : SubSubSystemButtonWidget('Overview'           , AxesRotationAxisTabs.OVERVIEW);
    button_processes        : SubSubSystemButtonWidget('Processes'          , AxesRotationAxisTabs.PROCESSES);
    button_driveChannel     : SubSubSystemButtonWidget('Drive channel'      , AxesRotationAxisTabs.DRIVE_CHANNEL);   
    button_virtualAxis      : SubSubSystemButtonWidget('Virtual axis'       , AxesRotationAxisTabs.VIRTUAL_AXIS);  
    button_physicalAxis     : SubSubSystemButtonWidget('Physical axis'      , AxesRotationAxisTabs.PHYSICAL_AXIS);  
    
    driveChannel    : AX52XXDriveChannelWidget;
    virtualAxis     : AngularAxisWidget;
    physicalAxis    : AngularAxisWidget;
    
    
    actPos : AxesAngleWidget;
    setPos : AxesAngleWidget;
    targetPos : AxesAngleWidget;
END_VAR


actualStatus(text  := ref.actualStatus,
             color := HealthBusyToColor(healthStatus := ref.statuses.healthStatus, 
                                        busyStatus   := ref.statuses.busyStatus));

processes_powerOffStatus(
    text  := ref.processes.powerOff.actualStatus,
    color := HealthBusyToColor(healthStatus := ref.processes.powerOff.statuses.healthStatus, 
                               busyStatus   := ref.processes.powerOff.statuses.busyStatus));
processes_powerOnStatus(
    text  := ref.processes.powerOn.actualStatus,
    color := HealthBusyToColor(healthStatus := ref.processes.powerOn.statuses.healthStatus, 
                               busyStatus   := ref.processes.powerOn.statuses.busyStatus));
processes_resetStatus(
    text  := ref.processes.reset.actualStatus,
    color := HealthBusyToColor(healthStatus := ref.processes.reset.statuses.healthStatus, 
                               busyStatus   := ref.processes.reset.statuses.busyStatus));
processes_stopStatus(
    text  := ref.processes.stop.actualStatus,
    color := HealthBusyToColor(healthStatus := ref.processes.stop.statuses.healthStatus, 
                               busyStatus   := ref.processes.stop.statuses.busyStatus));
processes_moveAbsoluteStatus(
    text  := ref.processes.moveAbsolute.actualStatus,
    color := HealthBusyToColor(healthStatus := ref.processes.moveAbsolute.statuses.healthStatus, 
                               busyStatus   := ref.processes.moveAbsolute.statuses.busyStatus));
processes_moveRelativeStatus(
    text  := ref.processes.moveRelative.actualStatus,
    color := HealthBusyToColor(healthStatus := ref.processes.moveRelative.statuses.healthStatus, 
                               busyStatus   := ref.processes.moveRelative.statuses.busyStatus));
processes_moveVelocityStatus(
    text  := ref.processes.moveVelocity.actualStatus,
    color := HealthBusyToColor(healthStatus := ref.processes.moveVelocity.statuses.healthStatus, 
                               busyStatus   := ref.processes.moveVelocity.statuses.busyStatus));
processes_moveOutOfLimitSwitchStatus(
    text  := ref.processes.moveOutOfLimitSwitch.actualStatus,
    color := HealthBusyToColor(healthStatus := ref.processes.moveOutOfLimitSwitch.statuses.healthStatus, 
                               busyStatus   := ref.processes.moveOutOfLimitSwitch.statuses.busyStatus));

driveChannel(ref := ref_driveChannel, name := driveChannelTitle);
virtualAxis(baseRef := ref.parts.virtualAxis, ref := ref.parts.virtualAxis);
physicalAxis(baseRef := ref.parts.physicalAxis, ref := ref.parts.physicalAxis);                

processCommonHealthStatus(
     isGood :=      ref.processes.powerOn.statuses.healthStatus.isGood 
                AND ref.processes.powerOff.statuses.healthStatus.isGood
                AND ref.processes.reset.statuses.healthStatus.isGood
                AND ref.processes.stop.statuses.healthStatus.isGood
                AND ref.processes.moveAbsolute.statuses.healthStatus.isGood
                AND ref.processes.moveRelative.statuses.healthStatus.isGood
                AND ref.processes.moveVelocity.statuses.healthStatus.isGood
                AND ref.processes.moveOutOfLimitSwitch.statuses.healthStatus.isGood,
     hasWarning :=  ref.processes.powerOn.statuses.healthStatus.hasWarning 
                 OR ref.processes.powerOff.statuses.healthStatus.hasWarning
                 OR ref.processes.reset.statuses.healthStatus.hasWarning
                 OR ref.processes.stop.statuses.healthStatus.hasWarning
                 OR ref.processes.moveAbsolute.statuses.healthStatus.hasWarning
                 OR ref.processes.moveRelative.statuses.healthStatus.hasWarning
                 OR ref.processes.moveVelocity.statuses.healthStatus.hasWarning
                 OR ref.processes.moveOutOfLimitSwitch.statuses.healthStatus.hasWarning);

processCommonBusyStatus(
    isBusy :=      ref.processes.powerOn.statuses.busyStatus.busy 
                 OR ref.processes.powerOff.statuses.busyStatus.busy
                 OR ref.processes.reset.statuses.busyStatus.busy
                 OR ref.processes.stop.statuses.busyStatus.busy
                 OR ref.processes.moveAbsolute.statuses.busyStatus.busy
                 OR ref.processes.moveRelative.statuses.busyStatus.busy
                 OR ref.processes.moveVelocity.statuses.busyStatus.busy
                 OR ref.processes.moveOutOfLimitSwitch.statuses.busyStatus.busy);

processCommonStatusColor := HealthBusyToColor(healthStatus := processCommonHealthStatus, busyStatus := processCommonBusyStatus);

button_overview(        color := actualStatus.color                     , activeTab := activeTab);
button_processes(       color := processCommonStatusColor               , activeTab := activeTab);
button_driveChannel(    color := driveChannel.actualStatus.color        , activeTab := activeTab);
button_virtualAxis(     color := virtualAxis.base.actualStatus.color    , activeTab := activeTab);
button_physicalAxis(    color := physicalAxis.base.actualStatus.color   , activeTab := activeTab);

actPos(degrees := ref.actPos.degrees.value, format := '%d° %.2d$' %04.1f"', showPlus := FALSE, showMinus := TRUE);
setPos(degrees := ref.setPos.degrees.value, format := '%d° %.2d$' %04.1f"', showPlus := FALSE, showMinus := TRUE);
targetPos(degrees := ref.targetPos.degrees.value, format := '%d° %.2d$' %04.1f"', showPlus := FALSE, showMinus := TRUE);

END_FUNCTION_BLOCK

// ---- MTCS/Axes/Widgets/AxesImageWidget.TcPOU
FUNCTION_BLOCK AxesImageWidget
VAR_INPUT
END_VAR
VAR_OUTPUT
    azi : LREAL;
    ele : LREAL;
    roc : LREAL;
    ron : LREAL;
    aziTopTubShown : INT;
    aziTarget : LREAL;
    eleTarget : LREAL;
    rocTarget : LREAL;
    ronTarget : LREAL;
    aziTargetInvisible : BOOL;
    eleTargetInvisible : BOOL;
    rocTargetInvisible : BOOL;
    ronTargetInvisible : BOOL;
    ronName : STRING;
    rocName : STRING;
    rocStationName : STRING;
    ronStationName : STRING;
END_VAR
VAR_IN_OUT
	ref : Axes;
END_VAR
VAR
    mark10Degrees : LREAL := 10; // used to make a 'mark' every 10 degrees on the graphical telescope image
    
END_VAR

azi := ref.parts.azi.actPos.degrees.value;
ele := ref.parts.ele.actPos.degrees.value - 90.0;
roc := - (ref.parts.roc.actPos.degrees.value + ref.config.rocGuiAngle);
ron := - (ref.parts.ron.actPos.degrees.value + ref.config.ronGuiAngle);
aziTarget := ref.target.aziPos.degrees.value;
eleTarget := ref.target.elePos.degrees.value - 90.0;
rocTarget := ref.target.paPos.degrees.value * ref.config.rocPositionAngleSign;
ronTarget := ref.target.paPos.degrees.value * ref.config.ronPositionAngleSign;
rocName := ref.config.cassegrainRotatorName;
ronName := ref.config.nasmythRotatorName;
rocStationName := 'Cassegrain';
ronStationName := 'Nasmyth';


aziTargetInvisible := NOT(ref.target.isValid AND ref.target.isGiven);
eleTargetInvisible := NOT(ref.target.isValid AND ref.target.isGiven);
rocTargetInvisible := NOT(ref.target.isValid AND ref.target.isGiven);
ronTargetInvisible := NOT(ref.target.isValid AND ref.target.isGiven);

IF ref.parts.ele.actPos.degrees.value > 87 THEN
    aziTopTubShown := 0;
ELSIF ref.parts.ele.actPos.degrees.value > 84 THEN
    aziTopTubShown := 1;
ELSIF ref.parts.ele.actPos.degrees.value > 78 THEN
    aziTopTubShown := 2;
ELSIF ref.parts.ele.actPos.degrees.value > 72 THEN
    aziTopTubShown := 3;
ELSIF ref.parts.ele.actPos.degrees.value > 66 THEN
    aziTopTubShown := 4;
ELSIF ref.parts.ele.actPos.degrees.value > 60 THEN
    aziTopTubShown := 5;
ELSIF ref.parts.ele.actPos.degrees.value > 54 THEN
    aziTopTubShown := 6;
ELSIF ref.parts.ele.actPos.degrees.value > 48 THEN
    aziTopTubShown := 7;
ELSIF ref.parts.ele.actPos.degrees.value > 42 THEN
    aziTopTubShown := 8;
ELSIF ref.parts.ele.actPos.degrees.value > 35 THEN
    aziTopTubShown := 9;
ELSIF ref.parts.ele.actPos.degrees.value > 28 THEN
    aziTopTubShown := 10;
ELSIF ref.parts.ele.actPos.degrees.value > 22 THEN
    aziTopTubShown := 11;
ELSIF ref.parts.ele.actPos.degrees.value > 17 THEN
    aziTopTubShown := 12;
ELSIF ref.parts.ele.actPos.degrees.value > 12 THEN
    aziTopTubShown := 13;
ELSE
    aziTopTubShown := 14;
END_IF

END_FUNCTION_BLOCK

// ---- MTCS/Axes/Widgets/AxesManualWidget.TcPOU
FUNCTION_BLOCK AxesManualWidget
VAR_INPUT

    activeTab : AxesManualTabs := AxesManualTabs.TAB_POSITIONS;

    joystickAziEle : AxesManualJoystickAziEleWidget;
    joystickRot : AxesManualJoystickRotWidget;
    offsets : AxesManualOffsetsWidget;
    positions : AxesManualPositionsWidget;
    moveAbsolute : AxesManualMoveAbsoluteWidget;
    moveVelocity : AxesManualMoveVelocityWidget;
END_VAR
VAR_OUTPUT
END_VAR
VAR_IN_OUT
    ref : Axes;
    ref_operatorStatus : OperatorStatus;
END_VAR
VAR
END_VAR

joystickAziEle(ref := ref);
joystickRot(ref := ref);
offsets(ref := ref);
positions(ref := ref, ref_operatorStatus := ref_operatorStatus);
moveAbsolute(ref := ref);
moveVelocity(ref := ref);

END_FUNCTION_BLOCK

// ---- MTCS/Axes/Widgets/AxesIOWidget.TcPOU
FUNCTION_BLOCK AxesIOWidget
VAR_INPUT
END_VAR
VAR_OUTPUT
END_VAR
VAR
	actualStatus : StatusWidget;
END_VAR
VAR_IN_OUT
	ref : AxesIO;
END_VAR

actualStatus(text  := ref.actualStatus,
             color := HealthToColor(ref.statuses.healthStatus));

END_FUNCTION_BLOCK

// ---- MTCS/Axes/Widgets/AxesPointingModelSetupWidget.TcPOU
FUNCTION_BLOCK AxesPointingModelSetupWidget
VAR_INPUT
    part : INT;
    enableButtonPressed : BOOL;
    disableButtonPressed : BOOL;
END_VAR
VAR_OUTPUT
    enableButtonDisabled : BOOL;
    disableButtonDisabled : BOOL;
END_VAR
VAR
    configManager : ConfigManagerWidget;
END_VAR
VAR_IN_OUT
	ref : AxesPointingModelSetup;
    ref_enable : AxesEnablePointingModelProcess;
    ref_disable : Process;
END_VAR

configManager(mgr := ref.parts.configManager);

IF enableButtonPressed THEN
    ref_enable.request(name := ref.config.name);
    enableButtonPressed := FALSE;
END_IF

IF disableButtonPressed THEN
    ref_disable.request();
    disableButtonPressed := FALSE;
END_IF

enableButtonDisabled := ref_enable.statuses.enabledStatus.disabled OR ref.config.name = '';
disableButtonDisabled := ref_disable.statuses.enabledStatus.disabled;

END_FUNCTION_BLOCK

// ---- MTCS/Common/Widgets/ConfigManagerWidget.TcPOU
FUNCTION_BLOCK ConfigManagerWidget
VAR_INPUT
END_VAR
VAR_OUTPUT
    actualStatus : StatusWidget;
    load : ReadXmlProcessWidget;
    save : WriteXmlProcessWidget;
END_VAR
VAR_IN_OUT
    mgr : ConfigManager;
END_VAR
VAR
END_VAR

actualStatus(
    text  := mgr.actualStatus,
    color := HealthBusyToColor(
        healthStatus := mgr.statuses.healthStatus,
        busyStatus := mgr.statuses.busyStatus));

load(process := mgr.processes.load);
save(process := mgr.processes.save);

END_FUNCTION_BLOCK

// ---- MTCS/Common/Widgets/ReadXmlProcessWidget.TcPOU
FUNCTION_BLOCK ReadXmlProcessWidget
VAR_INPUT
END_VAR
VAR_OUTPUT
	fgColor : DWORD;
	bgColor : DWORD;
	description : STRING;
END_VAR
VAR_IN_OUT
	process : ReadXmlProcess;
END_VAR
VAR
END_VAR

IF process.statuses.healthStatus.good THEN

	IF process.statuses.busyStatus.idle THEN
		fgColor := Colors.BLACK;
		bgColor := Colors.GREEN;
		description := 'Idle';
	ELSIF process.statuses.busyStatus.busy THEN
		fgColor := Colors.WHITE;
		bgColor := Colors.BLUE;
		description := 'Reading file...';
	ELSE
		fgColor := Colors.WHITE;
		bgColor := Colors.BLACK;
		description := '';
	END_IF;

ELSIF process.statuses.healthStatus.bad THEN
	
	fgColor := Colors.WHITE;
	bgColor := Colors.RED;
		
	IF process.statuses.busyStatus.idle THEN
		IF process.errorId = 0 THEN
			description := 'Error';
		ELSIF process.errorId = 1804 THEN
			description := 'Dirs/files not found';
		ELSE
			description := CONCAT(CONCAT('Error (', UDINT_TO_STRING(process.errorId)), ')');
		END_IF
	ELSIF process.statuses.busyStatus.busy THEN
		IF process.errorId = 0 THEN
			description := 'Busy and error';
		ELSE
			description := CONCAT(CONCAT('Busy and error (', UDINT_TO_STRING(process.errorId)), ')');
		END_IF
	ELSE
		IF process.errorId = 0 THEN
			description := 'Error';
		ELSE
			description := CONCAT(CONCAT('Error (', UDINT_TO_STRING(process.errorId)), ')');
		END_IF
	END_IF;

ELSE
	fgColor := Colors.WHITE;
	bgColor := Colors.BLACK;
	description := '';
END_IF;

END_FUNCTION_BLOCK

// ---- MTCS/Common/Widgets/WriteXmlProcessWidget.TcPOU
FUNCTION_BLOCK WriteXmlProcessWidget
VAR_INPUT
END_VAR
VAR_OUTPUT
	fgColor : DWORD;
	bgColor : DWORD;
	description : STRING;
END_VAR
VAR_IN_OUT
	process : WriteXmlProcess;
END_VAR
VAR
END_VAR

IF process.statuses.healthStatus.good THEN

	IF process.statuses.busyStatus.idle THEN
		fgColor := Colors.BLACK;
		bgColor := Colors.GREEN;
		description := 'Idle';
	ELSIF process.statuses.busyStatus.busy THEN
		fgColor := Colors.WHITE;
		bgColor := Colors.BLUE;
		description := 'Writing file...';
	ELSE
		fgColor := Colors.WHITE;
		bgColor := Colors.BLACK;
		description := '';
	END_IF;

ELSIF process.statuses.healthStatus.bad THEN
	
	fgColor := Colors.WHITE;
	bgColor := Colors.RED;
		
	IF process.statuses.busyStatus.idle THEN
		IF process.errorId = 0 THEN
			description := 'Error';
		ELSIF process.errorId = 1804 THEN
			description := 'Dirs/files not found';
		ELSE
			description := CONCAT(CONCAT('Error (', UDINT_TO_STRING(process.errorId)), ')');
		END_IF
	ELSIF process.statuses.busyStatus.busy THEN
		IF process.errorId = 0 THEN
			description := 'Busy and error';
		ELSE
			description := CONCAT(CONCAT('Busy and error (', UDINT_TO_STRING(process.errorId)), ')');
		END_IF
	ELSE
		IF process.errorId = 0 THEN
			description := 'Error';
		ELSE
			description := CONCAT(CONCAT('Error (', UDINT_TO_STRING(process.errorId)), ')');
		END_IF
	END_IF;

ELSE
	fgColor := Colors.WHITE;
	bgColor := Colors.BLACK;
	description := '';
END_IF;

END_FUNCTION_BLOCK

// ---- MTCS/Axes/Widgets/AxesPointingModelsSetupWidget.TcPOU
FUNCTION_BLOCK AxesPointingModelsSetupWidget
VAR_INPUT
    activeModel : INT;
END_VAR
VAR_OUTPUT
END_VAR
VAR
	actualStatus : StatusWidget;
    
    model0 : AxesPointingModelSetupWidget;
    model1 : AxesPointingModelSetupWidget;
    model2 : AxesPointingModelSetupWidget;
    model3 : AxesPointingModelSetupWidget;
    model4 : AxesPointingModelSetupWidget;
    model5 : AxesPointingModelSetupWidget;
    model6 : AxesPointingModelSetupWidget;
    model7 : AxesPointingModelSetupWidget;
    model8 : AxesPointingModelSetupWidget;
    model9 : AxesPointingModelSetupWidget;
END_VAR
VAR_IN_OUT
	ref : AxesPointingModelsSetup;
    ref_enable : AxesEnablePointingModelProcess;
    ref_disable : Process;
END_VAR

actualStatus(text  := ref.actualStatus,
             color := HealthBusyToColor(
                        healthStatus := ref.statuses.healthStatus, 
                        busyStatus   := ref.statuses.busyStatus));

model0(ref := ref.parts.model0, ref_enable := ref_enable, ref_disable := ref_disable);
model1(ref := ref.parts.model1, ref_enable := ref_enable, ref_disable := ref_disable);
model2(ref := ref.parts.model2, ref_enable := ref_enable, ref_disable := ref_disable);
model3(ref := ref.parts.model3, ref_enable := ref_enable, ref_disable := ref_disable);
model4(ref := ref.parts.model4, ref_enable := ref_enable, ref_disable := ref_disable);
model5(ref := ref.parts.model5, ref_enable := ref_enable, ref_disable := ref_disable);
model6(ref := ref.parts.model6, ref_enable := ref_enable, ref_disable := ref_disable);
model7(ref := ref.parts.model7, ref_enable := ref_enable, ref_disable := ref_disable);
model8(ref := ref.parts.model8, ref_enable := ref_enable, ref_disable := ref_disable);
model9(ref := ref.parts.model9, ref_enable := ref_enable, ref_disable := ref_disable);

END_FUNCTION_BLOCK

// ---- MTCS/Axes/Widgets/AxesSetTargetDialogWidget.TcPOU
FUNCTION_BLOCK AxesSetTargetDialogWidget
VAR_INPUT
    do_request : BOOL;
    field_alpha_h       : LREAL;
    field_alpha_m       : LREAL;
    field_alpha_s       : LREAL;
    field_alpha_decimal : LREAL;
    units_alpha         : AxesDialogAlphaUnits;
    field_delta_sign    : AxesDialogSign;
    field_delta_d       : LREAL;
    field_delta_m       : LREAL;
    field_delta_s       : LREAL;
    field_delta_decimal : LREAL;
    units_delta         : AxesDialogDeltaUnits;
    field_muAlpha       : LREAL;
    field_muDelta       : LREAL;
    units_mu            : AxesMuUnits;
    field_parallax      : LREAL;
    field_radialVelocity: LREAL;
    field_epoch         : LREAL := 2000.0;
END_VAR
VAR_OUTPUT
END_VAR
VAR_IN_OUT
    process : AxesSetTargetProcess;
END_VAR
VAR
    alpha : LREAL;
    alphaUnits : AxesAlphaUnits;
    delta : LREAL;
    deltaUnits : AxesDeltaUnits;
END_VAR

IF do_request THEN
    do_request := FALSE;
    
    CASE units_alpha OF
        AxesDialogAlphaUnits.DIALOG_HMS:
            alphaUnits := AxesAlphaUnits.DEGREES;
            alpha := HMS_TO_DEG(
                positive := TRUE,
                hours    := field_alpha_h,
                minutes  := field_alpha_m,
                seconds  := field_alpha_s);
        AxesDialogAlphaUnits.DIALOG_HOURS:
            alphaUnits := AxesAlphaUnits.HOURS;
            alpha := field_alpha_decimal;
        AxesDialogAlphaUnits.DIALOG_RADIANS:
            alphaUnits := AxesAlphaUnits.RADIANS;
            alpha := field_alpha_decimal;
	END_CASE
    
    CASE units_delta OF
        AxesDialogDeltaUnits.DIALOG_DMS:
            deltaUnits := AxesDeltaUnits.DEGREES;
            delta := DMS_TO_DEG(
                positive := field_delta_sign = AxesDialogSign.DIALOG_PLUS,
                degrees  := field_delta_d,
                minutes  := field_delta_m,
                seconds  := field_delta_s);
        AxesDialogDeltaUnits.DIALOG_DEGREES:
            deltaUnits := AxesDeltaUnits.DEGREES;
            delta := field_delta_decimal;
        AxesDialogDeltaUnits.DIALOG_RADIANS:
            deltaUnits := AxesDeltaUnits.RADIANS;
            delta := field_delta_decimal;
	END_CASE
    
    CASE units_delta OF
        AxesDialogDeltaUnits.DIALOG_DMS:
            deltaUnits := AxesDeltaUnits.DEGREES;
            delta := DMS_TO_DEG(
                positive := field_delta_sign = AxesDialogSign.DIALOG_PLUS,
                degrees  := field_delta_d,
                minutes  := field_delta_m,
                seconds  := field_delta_s);
        AxesDialogDeltaUnits.DIALOG_RADIANS:
            deltaUnits := AxesDeltaUnits.RADIANS;
            delta := field_delta_decimal;
	END_CASE
    
    process.request(
        alpha           := alpha,
        alphaUnits      := alphaUnits,
        delta           := delta,
        deltaUnits      := deltaUnits,
        muUnits         := units_mu,
        muAlpha         := field_muAlpha,
        muDelta         := field_muDelta,
        parallax        := field_parallax,
        radialVelocity  := field_radialVelocity,
        epoch           := field_epoch);

END_IF

END_FUNCTION_BLOCK

// ---- MTCS/Axes/Widgets/AxesPointDialogWidget.TcPOU
FUNCTION_BLOCK AxesPointDialogWidget
VAR_INPUT
    do_request : BOOL;
    field_alpha_h       : LREAL;
    field_alpha_m       : LREAL;
    field_alpha_s       : LREAL;
    field_alpha_decimal : LREAL;
    units_alpha         : AxesDialogAlphaUnits;
    field_delta_sign    : AxesDialogSign;
    field_delta_d       : LREAL;
    field_delta_m       : LREAL;
    field_delta_s       : LREAL;
    field_delta_decimal : LREAL;
    units_delta         : AxesDialogDeltaUnits;
    field_muAlpha       : LREAL;
    field_muDelta       : LREAL;
    units_mu            : AxesMuUnits;
    field_parallax      : LREAL;
    field_radialVelocity: LREAL;
    field_epoch         : LREAL := 2000.0;
    field_tracking      : BOOL := TRUE;
    
    
    units_rot           : AxesMoveProcessWidgetUnits;
    
    
    field_rot_decimal   : LREAL;
    field_rot_sign      : AxesDialogSign;
    field_rot_d         : LREAL;
    field_rot_m         : LREAL;
    field_rot_s         : LREAL;
    
    field_roc_decimal   : LREAL;
    field_roc_sign      : AxesDialogSign;
    field_roc_d         : LREAL;
    field_roc_m         : LREAL;
    field_roc_s         : LREAL;
    
    field_ron_decimal   : LREAL;
    field_ron_sign      : AxesDialogSign;
    field_ron_d         : LREAL;
    field_ron_m         : LREAL;
    field_ron_s         : LREAL;
    
    selected_rot : BOOL;
    selected_ron : BOOL;
    selected_roc : BOOL;
    
END_VAR
VAR_OUTPUT
END_VAR
VAR_IN_OUT
    process : AxesPointProcess;
END_VAR
VAR
    alpha : LREAL;
    alphaUnits : AxesAlphaUnits;
    delta : LREAL;
    deltaUnits : AxesDeltaUnits;
    rotDeg : LREAL;
    ronDeg : LREAL;
    rocDeg : LREAL;
END_VAR

IF do_request THEN
    do_request := FALSE;
    
    CASE units_alpha OF
        AxesDialogAlphaUnits.DIALOG_HMS:
            alphaUnits := AxesAlphaUnits.DEGREES;
            alpha := HMS_TO_DEG(
                positive := TRUE,
                hours    := field_alpha_h,
                minutes  := field_alpha_m,
                seconds  := field_alpha_s);
        AxesDialogAlphaUnits.DIALOG_HOURS:
            alphaUnits := AxesAlphaUnits.HOURS;
            alpha := field_alpha_decimal;
        AxesDialogAlphaUnits.DIALOG_RADIANS:
            alphaUnits := AxesAlphaUnits.RADIANS;
            alpha := field_alpha_decimal;
	END_CASE
    
    CASE units_delta OF
        AxesDialogDeltaUnits.DIALOG_DMS:
            deltaUnits := AxesDeltaUnits.DEGREES;
            delta := DMS_TO_DEG(
                positive := field_delta_sign = AxesDialogSign.DIALOG_PLUS,
                degrees  := field_delta_d,
                minutes  := field_delta_m,
                seconds  := field_delta_s);
        AxesDialogDeltaUnits.DIALOG_DEGREES:
            deltaUnits := AxesDeltaUnits.DEGREES;
            delta := field_delta_decimal;
        AxesDialogDeltaUnits.DIALOG_RADIANS:
            deltaUnits := AxesDeltaUnits.RADIANS;
            delta := field_delta_decimal;
	END_CASE
    
    CASE units_rot OF
        AxesMoveProcessWidgetUnits.ARCMINUTES:
            rotDeg := field_rot_decimal / 60.0;
            rocDeg := field_roc_decimal / 60.0;
            ronDeg := field_ron_decimal / 60.0;
        AxesMoveProcessWidgetUnits.ARCSECCONDS:
            rotDeg := field_rot_decimal / 3600.0;
            rocDeg := field_roc_decimal / 3600.0;
            ronDeg := field_ron_decimal / 3600.0;
        AxesMoveProcessWidgetUnits.DEGMINSEC:
            rotDeg := DMS_TO_DEG(
                positive := field_rot_sign = AxesDialogSign.DIALOG_PLUS,
                degrees  := field_rot_d,
                minutes  := field_rot_m,
                seconds  := field_rot_s);
            rocDeg := DMS_TO_DEG(
                positive := field_roc_sign = AxesDialogSign.DIALOG_PLUS,
                degrees  := field_roc_d,
                minutes  := field_roc_m,
                seconds  := field_roc_s);
            ronDeg := DMS_TO_DEG(
                positive := field_ron_sign = AxesDialogSign.DIALOG_PLUS,
                degrees  := field_ron_d,
                minutes  := field_ron_m,
                seconds  := field_ron_s);
        AxesMoveProcessWidgetUnits.DEGREES:
            rotDeg := field_rot_decimal;
            rocDeg := field_roc_decimal;
            ronDeg := field_ron_decimal;
        AxesMoveProcessWidgetUnits.RADIANS:
            rotDeg := RAD_TO_DEG(field_rot_decimal);
            rocDeg := RAD_TO_DEG(field_roc_decimal);
            ronDeg := RAD_TO_DEG(field_ron_decimal);
    END_CASE

    
    
    
    
    process.request(
        alpha           := alpha,
        alphaUnits      := alphaUnits,
        delta           := delta,
        deltaUnits      := deltaUnits,
        muUnits         := units_mu,
        muAlpha         := field_muAlpha,
        muDelta         := field_muDelta,
        parallax        := field_parallax,
        radialVelocity  := field_radialVelocity,
        epoch           := field_epoch,
        tracking        := field_tracking,
        rotUnits        := AxesMoveUnits.DEGREES,
        rotOffset       := rotDeg,
        rocOffset       := rocDeg,
        ronOffset       := ronDeg,
        doRotOffset     := selected_rot,
        doRocOffset     := selected_roc,
        doRonOffset     := selected_ron);
END_IF

END_FUNCTION_BLOCK

// ---- MTCS/Axes/Widgets/AxesTargetWidget.TcPOU
FUNCTION_BLOCK AxesTargetWidget
VAR_INPUT
END_VAR
VAR_OUTPUT
	actualStatus : StatusWidget;
    alpha : AxesAlphaWidget;
    delta : AxesDeltaWidget;
    aziPos : AxesAngleWidget;
    elePos : AxesAngleWidget;
    paPos : AxesAngleWidget;
    
    alphaString : STRING;
    deltaString : STRING;
    aziString : STRING;
    eleString : STRING;
    paString : STRING;
END_VAR
VAR_IN_OUT
    ref : AxesTarget;
END_VAR
VAR
END_VAR

actualStatus(text  := ref.actualStatus,
             color := HealthToColor(healthStatus := ref.statuses.healthStatus));
                                        
alpha(radians := ref.alpha.radians.value);
delta(radians := ref.delta.radians.value);




aziPos(degrees := ref.aziPos.degrees.value, showPlus := FALSE, showMinus := TRUE);
elePos(degrees := ref.elePos.degrees.value, showPlus := TRUE, showMinus := TRUE);
paPos(degrees := ref.paPos.degrees.value, showPlus := TRUE, showMinus := TRUE);

IF ref.isGiven THEN
    alphaString := alpha.hmsString;
    deltaString := delta.dmsString;
    aziString := aziPos.dmsString;
    eleString := elePos.dmsString;
    paString := paPos.dmsString;
ELSE
    alphaString := '';
    deltaString := '';
    aziString := '';
    eleString := '';
    paString := '';
END_IF

END_FUNCTION_BLOCK

// ---- MTCS/Axes/Widgets/AxesFeedbackWidget.TcPOU
FUNCTION_BLOCK AxesFeedbackWidget
VAR_INPUT
END_VAR
VAR_OUTPUT
	actualStatus : StatusWidget;
    alpha : AxesAlphaWidget;
    delta : AxesDeltaWidget;
    
    aziPos : AxesAngleWidget;
    elePos : AxesAngleWidget;
    rocPos : AxesAngleWidget;
    ronPos : AxesAngleWidget;
END_VAR
VAR_IN_OUT
    ref : AxesFeedback;
END_VAR
VAR
END_VAR

actualStatus(text  := ref.actualStatus,
             color := HealthToColor(healthStatus := ref.statuses.healthStatus));

alpha(radians := ref.alpha.radians.value);
delta(radians := ref.delta.radians.value);


aziPos(degrees := ref.aziPos.degrees.value, showPlus := FALSE, showMinus := TRUE);
elePos(degrees := ref.elePos.degrees.value, showPlus := TRUE, showMinus := TRUE);
rocPos(degrees := ref.rocPos.degrees.value, showPlus := TRUE, showMinus := TRUE);
ronPos(degrees := ref.ronPos.degrees.value, showPlus := TRUE, showMinus := TRUE);

END_FUNCTION_BLOCK

// ---- MTCS/Axes/Widgets/AxesWidget.TcPOU
FUNCTION_BLOCK AxesWidget
VAR_INPUT
    activeTab : AxesTabs := AxesTabs.OVERVIEW;
    activeConfigTab : INT;
    activeConfigPosition : INT;
    
END_VAR
VAR_OUTPUT
    configManager           : ConfigManagerWidget;
	actualStatus            : StatusWidget;
	initializationStatus    : InitializationStatusWidget;
    isDerotatorActive : BOOL;
    name : STRING := 'Axes';
END_VAR
VAR_IN_OUT
	ref : Axes;
    ref_operatorStatus : OperatorStatus;
END_VAR
VAR
    axes : AxesAxesWidget;
    tpoint : AxesPointingModelsSetupWidget;
    io : AxesIOWidget;
    image : AxesImageWidget;
    target : AxesTargetWidget;
    feedback : AxesFeedbackWidget;

    manual : AxesManualWidget;
    
    button_initialize : InitializeButtonWidget;
    button_operating  : OperatingButtonWidget;
    button_locking    : LockingButtonWidget;
    
    button_overview         : SubSystemButtonWidget('Overview'	, AxesTabs.OVERVIEW);
    button_manual           : SubSystemButtonWidget('Manual'    , Axestabs.MANUAL);
    button_axes             : SubSystemButtonWidget('Axes'      , AxesTabs.AXES);
    button_target           : SubSystemButtonWidget('Target'    , Axestabs.TARGET);
    button_tpoint           : SubSystemButtonWidget('TPoint'  	, AxesTabs.TPOINT);
    button_advanced         : SubSystemButtonWidget('Advanced'  , AxesTabs.ADVANCED);
    button_io               : SubSystemButtonWidget('I/O'     	, Axestabs.IO);
    button_config           : SubSystemButtonWidget('Config'  	, AxesTabs.CONFIG);
    
    
    cppAxesErrorString : STRING;
    
    targetHealthStatus : HealthStatus;
    
    quickElevation : AxesAngleWidget;
    last : AxesAlphaWidget;
    ha : AxesAlphaWidget;
    
    setTarget : AxesSetTargetDialogWidget;
    point : AxesPointDialogWidget;
    
    activePointingModelString : STRING;
    activeRotatorString : STRING;
    
    processes_powerOnStatus : StatusWidget;
    processes_powerOffStatus : StatusWidget;
    processes_resetStatus : StatusWidget;
    processes_doHomingStatus : StatusWidget;
    processes_stopStatus : StatusWidget;
    processes_quickStopStatus : StatusWidget;
    processes_pointStatus : StatusWidget;
    
    processes_powerOnArgs : AxesMultiPowerOnProcessArgs;
END_VAR

initializationStatus(status := ref.statuses.initializationStatus);
configManager(mgr := ref.parts.configManager);
axes(ref_azi := ref.parts.azi,
     ref_ele := ref.parts.ele,
     ref_roc := ref.parts.roc,
     ref_ron := ref.parts.ron,
     ref_io  := ref.parts.io); // TODO
tpoint(ref          := ref.parts.tpoint, 
       ref_enable   := ref.processes.enablePointingModel, 
       ref_disable  := ref.processes.disablePointingModel);
io(ref := ref.parts.io);
image(ref := ref);
manual(ref := ref, ref_operatorStatus := ref_operatorStatus);
target(ref := ref.target);
feedback(ref := ref.feedback);

targetHealthStatus(isGood := ref.fromCppAxes.error = TmcAxesErrors.AXES_NO_ERROR);
isDerotatorActive := ref.activeRotator <> AxesRotatorActivity.NONE_ACTIVE;

button_initialize(status := ref.statuses.initializationStatus, process := ref.processes.initialize);
button_operating(status := ref.statuses.operatingStatus, process := ref.processes.changeOperatingState);
button_locking(status := ref.statuses.initializationStatus, lock := ref.processes.lock, unlock := ref.processes.unlock);

button_overview(        color := actualStatus.color                 , activeTab := activeTab);
button_manual(          color := actualStatus.color                 , activeTab := activeTab);
button_axes(            color := axes.commonStatusColor             , activeTab := activeTab);
button_target(          color := HealthToColor(targetHealthStatus)  , activeTab := activeTab);
button_tpoint(          color := tpoint.actualStatus.color          , activeTab := activeTab);
button_advanced(        color := actualStatus.color                 , activeTab := activeTab);
button_io(              color := io.actualStatus.color              , activeTab := activeTab);
button_config(          color := configManager.actualStatus.color   , activeTab := activeTab);

actualStatus(text  := ref.actualStatus,
             color := SystemToColor(healthStatus := ref.statuses.healthStatus,
                                    busyStatus   := ref.statuses.busyStatus,
                                    initializationStatus := ref.statuses.initializationStatus,
                                    operatingStatus := ref.statuses.operatingStatus));

cppAxesErrorString := TmcAxesErrorsToString(ref.fromCppAxes.error);


ha(radians := ref.fromCppAxes.ha);
last(radians := ref.fromCppAxes.last);
quickElevation(degrees := RAD_TO_DEG(ref.fromCppAxes.object.quick.el));

// dialogs
setTarget(process := ref.processes.setTarget);
point(process := ref.processes.point);

IF ref.isPointingModelActive THEN
    activePointingModelString := ref.activePointingModel.name;
ELSE
    activePointingModelString := '';
END_IF

CASE ref.activeRotator OF
    AxesRotatorActivity.NONE_ACTIVE:
        activeRotatorString := 'None';
    AxesRotatorActivity.ROC_ACTIVE:
        activeRotatorString := CONCAT(ref.config.cassegrainRotatorName, ' (ROC)');
    AxesRotatorActivity.RON_ACTIVE:
        activeRotatorString := CONCAT(ref.config.cassegrainRotatorName, ' (RON)');
END_CASE


processes_powerOffStatus(
    text  := ref.processes.powerOff.actualStatus,
    color := HealthBusyToColor(healthStatus := ref.processes.powerOff.statuses.healthStatus, 
                               busyStatus   := ref.processes.powerOff.statuses.busyStatus));
processes_powerOnStatus(
    text  := ref.processes.powerOn.actualStatus,
    color := HealthBusyToColor(healthStatus := ref.processes.powerOn.statuses.healthStatus, 
                               busyStatus   := ref.processes.powerOn.statuses.busyStatus));

processes_resetStatus(
    text  := ref.processes.reset.actualStatus,
    color := HealthBusyToColor(healthStatus := ref.processes.reset.statuses.healthStatus, 
                               busyStatus   := ref.processes.reset.statuses.busyStatus));
processes_doHomingStatus(
    text  := ref.processes.doHoming.actualStatus,
    color := HealthBusyToColor(healthStatus := ref.processes.doHoming.statuses.healthStatus, 
                               busyStatus   := ref.processes.doHoming.statuses.busyStatus));            
processes_stopStatus(
    text  := ref.processes.stop.actualStatus,
    color := HealthBusyToColor(healthStatus := ref.processes.stop.statuses.healthStatus, 
                               busyStatus   := ref.processes.stop.statuses.busyStatus));        
processes_quickStopStatus(
    text  := ref.processes.quickStop.actualStatus,
    color := HealthBusyToColor(healthStatus := ref.processes.quickStop.statuses.healthStatus, 
                               busyStatus   := ref.processes.quickStop.statuses.busyStatus));    
processes_pointStatus(
    text  := ref.processes.point.actualStatus,
    color := HealthBusyToColor(healthStatus := ref.processes.point.statuses.healthStatus, 
                               busyStatus   := ref.processes.point.statuses.busyStatus));

END_FUNCTION_BLOCK

// ---- MTCS/Common/Widgets/InitializationStatusWidget.TcPOU
FUNCTION_BLOCK InitializationStatusWidget
VAR_INPUT
END_VAR
VAR_OUTPUT
	fgColor : DWORD;
	bgColor : DWORD;
	description : STRING;
END_VAR
VAR_IN_OUT
	status : InitializationStatus;
END_VAR
VAR
END_VAR

IF status.initialized THEN
	fgColor := Colors.BLACK;
	bgColor := Colors.GREEN;
	description := 'Initialized';
ELSIF status.initializing THEN
	fgColor := Colors.WHITE;
	bgColor := Colors.BLUE;
	description := 'Initializing';
ELSIF status.locked THEN
	fgColor := Colors.BLACK;
	bgColor := Colors.ORANGE;
	description := 'LOCKED';
ELSIF status.shutdown THEN
	fgColor := Colors.BLACK;
	bgColor := Colors.GRAY;
	description := 'Shutdown';
ELSIF status.initializingFailed THEN
	fgColor := Colors.WHITE;
	bgColor := Colors.RED;
	description := 'Failed';
ELSE
	fgColor := Colors.WHITE;
	bgColor := Colors.RED;
	description := 'Unknown';
END_IF

END_FUNCTION_BLOCK

// ---- MTCS/Common/Widgets/InitializeButtonWidget.TcPOU
FUNCTION_BLOCK InitializeButtonWidget
VAR_INPUT
END_VAR
VAR_OUTPUT
    text : STRING;
    textOneLine : STRING;
    deactivate : BOOL;
END_VAR
VAR_IN_OUT
    status : InitializationStatus;
	process : Process;
END_VAR
VAR
    do_request : BOOL := FALSE;
END_VAR

IF status.initialized THEN
    text := 'Re-$ninitialize';
    textOneLine := 'Reinitialize';
    deactivate := process.statuses.enabledStatus.disabled;
ELSIF status.initializing THEN
    text := 'Re-$ninitialize';
    textOneLine := 'Reinitialize';
    deactivate := process.statuses.enabledStatus.disabled;
ELSIF status.initializingFailed THEN
    text := 'Re-$ninitialize';
    textOneLine := 'Reinitialize';
    deactivate := process.statuses.enabledStatus.disabled;
ELSIF status.shutdown THEN
    text := 'Initialize';
    textOneLine := 'Initialize';
    deactivate := process.statuses.enabledStatus.disabled;
ELSE
    text := 'Re-$ninitialize';
    textOneLine := 'Reinitialize';
    deactivate := process.statuses.enabledStatus.disabled;
END_IF


IF do_request THEN
    process.request();
    do_request := FALSE;
END_IF

END_FUNCTION_BLOCK

